    // shielded helion to proton mag. mom. ratio
    // Uncertainty: 8.9e-09
    fShieldedHelionToProtonMag_Mom_Ratio : LREAL := -0.7617665618;
    fShieldedHelionToProtonMag_Mom_Ratio_Uncertainty : LREAL := 8.9e-09;

    // shielded helion to shielded proton mag. mom. ratio
    // Uncertainty: 3.3e-09
    fShieldedHelionToShieldedProtonMag_Mom_Ratio : LREAL := -0.7617861313;
    fShieldedHelionToShieldedProtonMag_Mom_Ratio_Uncertainty : LREAL := 3.3e-09;

    // shielded proton gyromag. ratio (s^-1 T^-1)
    // Uncertainty: 2.9
    fShieldedProtonGyromag_Ratio_in_s_1_T_1 : LREAL := 267515315.1;
    fShieldedProtonGyromag_Ratio_in_s_1_T_1_Units : STRING := 's^-1 T^-1';
    fShieldedProtonGyromag_Ratio_in_s_1_T_1_Uncertainty : LREAL := 2.9;

    // shielded proton gyromag. ratio over 2 pi (MHz T^-1)
    // Uncertainty: 5.3e-07
    fShieldedProtonGyromag_RatioOver2Pi_in_MHz_T_1 : LREAL := 42.57638507;
    fShieldedProtonGyromag_RatioOver2Pi_in_MHz_T_1_Units : STRING := 'MHz T^-1';
    fShieldedProtonGyromag_RatioOver2Pi_in_MHz_T_1_Uncertainty : LREAL := 5.3e-07;

    // shielded proton mag. mom. (J T^-1)
    // Uncertainty: 1.5e-34
    fShieldedProtonMag_Mom_in_J_T_1 : LREAL := 1.41057056e-26;
    fShieldedProtonMag_Mom_in_J_T_1_Units : STRING := 'J T^-1';
    fShieldedProtonMag_Mom_in_J_T_1_Uncertainty : LREAL := 1.5e-34;

    // shielded proton mag. mom. to Bohr magneton ratio
    // Uncertainty: 1.7e-11
    fShieldedProtonMag_Mom_ToBohrMagnetonRatio : LREAL := 0.001520993128;
    fShieldedProtonMag_Mom_ToBohrMagnetonRatio_Uncertainty : LREAL := 1.7e-11;

    // shielded proton mag. mom. to nuclear magneton ratio
    // Uncertainty: 3e-08
    fShieldedProtonMag_Mom_ToNuclearMagnetonRatio : LREAL := 2.792775599;
    fShieldedProtonMag_Mom_ToNuclearMagnetonRatio_Uncertainty : LREAL := 3e-08;

    // speed of light in vacuum (m s^-1)
    fSpeedOfLightInVacuum_in_m_s_1 : LREAL := 299792458.0;
    fSpeedOfLightInVacuum_in_m_s_1_Units : STRING := 'm s^-1';

    // standard acceleration of gravity (m s^-2)
    fStandardAccelerationOfGravity_in_m_s_2 : LREAL := 9.80665;
    fStandardAccelerationOfGravity_in_m_s_2_Units : STRING := 'm s^-2';

    // standard atmosphere (Pa)
    fStandardAtmosphere_in_Pa : LREAL := 101325.0;
    fStandardAtmosphere_in_Pa_Units : STRING := 'Pa';

    // Stefan-Boltzmann constant (W m^-2 K^-4)
    fStefan_BoltzmannConstant_in_W_m_2_K_4 : LREAL := 5.670374419e-08;
    fStefan_BoltzmannConstant_in_W_m_2_K_4_Units : STRING := 'W m^-2 K^-4';

    // tau Compton wavelength (m)
    // Uncertainty: 4.7e-20
    fTauComptonWavelength_in_m : LREAL := 6.97771e-16;
    fTauComptonWavelength_in_m_Units : STRING := 'm';
    fTauComptonWavelength_in_m_Uncertainty : LREAL := 4.7e-20;

    // tau Compton wavelength over 2 pi (m)
    // Uncertainty: 1e-20
    fTauComptonWavelengthOver2Pi_in_m : LREAL := 1.11056e-16;
    fTauComptonWavelengthOver2Pi_in_m_Units : STRING := 'm';
    fTauComptonWavelengthOver2Pi_in_m_Uncertainty : LREAL := 1e-20;

    // tau-electron mass ratio
    // Uncertainty: 0.23
    fTauElectronMassRatio : LREAL := 3477.23;
    fTauElectronMassRatio_Uncertainty : LREAL := 0.23;

    // tau mass (kg)
    // Uncertainty: 2.1e-31
    fTauMass_in_kg : LREAL := 3.16754e-27;
    fTauMass_in_kg_Units : STRING := 'kg';
    fTauMass_in_kg_Uncertainty : LREAL := 2.1e-31;

    // tau mass energy equivalent (J)
    // Uncertainty: 1.9e-14
    fTauMassEnergyEquivalent_in_J : LREAL := 2.84684e-10;
    fTauMassEnergyEquivalent_in_J_Units : STRING := 'J';
    fTauMassEnergyEquivalent_in_J_Uncertainty : LREAL := 1.9e-14;

    // tau mass energy equivalent in MeV (MeV)
    // Uncertainty: 0.16
    fTauMassEnergyEquivalentInMeV_in_MeV : LREAL := 1776.82;
    fTauMassEnergyEquivalentInMeV_in_MeV_Units : STRING := 'MeV';
    fTauMassEnergyEquivalentInMeV_in_MeV_Uncertainty : LREAL := 0.16;

    // tau mass in u (u)
    // Uncertainty: 0.00013
    fTauMassInU_in_u : LREAL := 1.90754;
    fTauMassInU_in_u_Units : STRING := 'u';
    fTauMassInU_in_u_Uncertainty : LREAL := 0.00013;

    // tau molar mass (kg mol^-1)
    // Uncertainty: 1.3e-07
    fTauMolarMass_in_kg_mol_1 : LREAL := 0.00190754;
    fTauMolarMass_in_kg_mol_1_Units : STRING := 'kg mol^-1';
    fTauMolarMass_in_kg_mol_1_Uncertainty : LREAL := 1.3e-07;

    // tau-muon mass ratio
    // Uncertainty: 0.0011
    fTauMuonMassRatio : LREAL := 16.817;
    fTauMuonMassRatio_Uncertainty : LREAL := 0.0011;

    // tau-neutron mass ratio
    // Uncertainty: 0.00013
    fTauNeutronMassRatio : LREAL := 1.89115;
    fTauNeutronMassRatio_Uncertainty : LREAL := 0.00013;

    // tau-proton mass ratio
    // Uncertainty: 0.00013
    fTauProtonMassRatio : LREAL := 1.89376;
    fTauProtonMassRatio_Uncertainty : LREAL := 0.00013;

    // Thomson cross section (m^2)
    // Uncertainty: 6e-38
    fThomsonCrossSection_in_m_2 : LREAL := 6.6524587321e-29;
    fThomsonCrossSection_in_m_2_Units : STRING := 'm^2';
    fThomsonCrossSection_in_m_2_Uncertainty : LREAL := 6e-38;

    // triton-electron mag. mom. ratio
    // Uncertainty: 2.1e-11
    fTritonElectronMag_Mom_Ratio : LREAL := -0.001620514423;
    fTritonElectronMag_Mom_Ratio_Uncertainty : LREAL := 2.1e-11;

    // triton-electron mass ratio
    // Uncertainty: 2.7e-07
    fTritonElectronMassRatio : LREAL := 5496.92153573;
    fTritonElectronMassRatio_Uncertainty : LREAL := 2.7e-07;

    // triton g factor
    // Uncertainty: 1.2e-08
    fTritonGFactor : LREAL := 5.957924931;
    fTritonGFactor_Uncertainty : LREAL := 1.2e-08;

    // triton mag. mom. (J T^-1)
    // Uncertainty: 3e-35
    fTritonMag_Mom_in_J_T_1 : LREAL := 1.5046095202e-26;
    fTritonMag_Mom_in_J_T_1_Units : STRING := 'J T^-1';
    fTritonMag_Mom_in_J_T_1_Uncertainty : LREAL := 3e-35;

    // triton mag. mom. to Bohr magneton ratio
    // Uncertainty: 3.2e-12
    fTritonMag_Mom_ToBohrMagnetonRatio : LREAL := 0.0016223936651;
    fTritonMag_Mom_ToBohrMagnetonRatio_Uncertainty : LREAL := 3.2e-12;

    // triton mag. mom. to nuclear magneton ratio
    // Uncertainty: 5.9e-09
    fTritonMag_Mom_ToNuclearMagnetonRatio : LREAL := 2.9789624656;
    fTritonMag_Mom_ToNuclearMagnetonRatio_Uncertainty : LREAL := 5.9e-09;

    // triton mass (kg)
    // Uncertainty: 1.5e-36
    fTritonMass_in_kg : LREAL := 5.0073567446e-27;
    fTritonMass_in_kg_Units : STRING := 'kg';
    fTritonMass_in_kg_Uncertainty : LREAL := 1.5e-36;

    // triton mass energy equivalent (J)
    // Uncertainty: 1.4e-19
    fTritonMassEnergyEquivalent_in_J : LREAL := 4.500387806e-10;
    fTritonMassEnergyEquivalent_in_J_Units : STRING := 'J';
    fTritonMassEnergyEquivalent_in_J_Uncertainty : LREAL := 1.4e-19;

    // triton mass energy equivalent in MeV (MeV)
    // Uncertainty: 8.5e-07
    fTritonMassEnergyEquivalentInMeV_in_MeV : LREAL := 2808.92113298;
    fTritonMassEnergyEquivalentInMeV_in_MeV_Units : STRING := 'MeV';
    fTritonMassEnergyEquivalentInMeV_in_MeV_Uncertainty : LREAL := 8.5e-07;

    // triton mass in u (u)
    // Uncertainty: 1.2e-10
    fTritonMassInU_in_u : LREAL := 3.01550071621;
    fTritonMassInU_in_u_Units : STRING := 'u';
    fTritonMassInU_in_u_Uncertainty : LREAL := 1.2e-10;

    // triton molar mass (kg mol^-1)
    // Uncertainty: 9.2e-13
    fTritonMolarMass_in_kg_mol_1 : LREAL := 0.00301550071517;
    fTritonMolarMass_in_kg_mol_1_Units : STRING := 'kg mol^-1';
    fTritonMolarMass_in_kg_mol_1_Uncertainty : LREAL := 9.2e-13;

    // triton-neutron mag. mom. ratio
    // Uncertainty: 3.7e-07
    fTritonNeutronMag_Mom_Ratio : LREAL := -1.55718553;
    fTritonNeutronMag_Mom_Ratio_Uncertainty : LREAL := 3.7e-07;

    // triton-proton mag. mom. ratio
    // Uncertainty: 1e-08
    fTritonProtonMag_Mom_Ratio : LREAL := 1.066639908;
    fTritonProtonMag_Mom_Ratio_Uncertainty : LREAL := 1e-08;

    // triton-proton mass ratio
    // Uncertainty: 1.5e-10
    fTritonProtonMassRatio : LREAL := 2.99371703414;
    fTritonProtonMassRatio_Uncertainty : LREAL := 1.5e-10;

    // unified atomic mass unit (kg)
    // Uncertainty: 5e-37
    fUnifiedAtomicMassUnit_in_kg : LREAL := 1.6605390666e-27;
    fUnifiedAtomicMassUnit_in_kg_Units : STRING := 'kg';
    fUnifiedAtomicMassUnit_in_kg_Uncertainty : LREAL := 5e-37;

    // von Klitzing constant (ohm)
    fVonKlitzingConstant_in_ohm : LREAL := 25812.80745;
    fVonKlitzingConstant_in_ohm_Units : STRING := 'ohm';

    // weak mixing angle
    // Uncertainty: 0.0003
    fWeakMixingAngle : LREAL := 0.2229;
    fWeakMixingAngle_Uncertainty : LREAL := 0.0003;

    // Wien frequency displacement law constant (Hz K^-1)
    fWienFrequencyDisplacementLawConstant_in_Hz_K_1 : LREAL := 58789257570.0;
    fWienFrequencyDisplacementLawConstant_in_Hz_K_1_Units : STRING := 'Hz K^-1';

    // Wien wavelength displacement law constant (m K)
    fWienWavelengthDisplacementLawConstant_in_m_K : LREAL := 0.002897771955;
    fWienWavelengthDisplacementLawConstant_in_m_K_Units : STRING := 'm K';

    // atomic unit of mom.um (kg m s^-1)
    // Uncertainty: 2.4e-32
    fAtomicUnitOfMom_um_in_kg_m_s_1 : LREAL := 1.992851882e-24;
    fAtomicUnitOfMom_um_in_kg_m_s_1_Units : STRING := 'kg m s^-1';
    fAtomicUnitOfMom_um_in_kg_m_s_1_Uncertainty : LREAL := 2.4e-32;

    // electron-helion mass ratio
    // Uncertainty: 7.9e-15
    fElectronHelionMassRatio : LREAL := 0.0001819543074573;
    fElectronHelionMassRatio_Uncertainty : LREAL := 7.9e-15;

    // electron-triton mass ratio
    // Uncertainty: 9e-15
    fElectronTritonMassRatio : LREAL := 0.0001819200062251;
    fElectronTritonMassRatio_Uncertainty : LREAL := 9e-15;

    // helion g factor
    // Uncertainty: 5e-08
    fHelionGFactor : LREAL := -4.255250615;
    fHelionGFactor_Uncertainty : LREAL := 5e-08;

    // helion mag. mom. (J T^-1)
    // Uncertainty: 1.3e-34
    fHelionMag_Mom_in_J_T_1 : LREAL := -1.074617532e-26;
    fHelionMag_Mom_in_J_T_1_Units : STRING := 'J T^-1';
    fHelionMag_Mom_in_J_T_1_Uncertainty : LREAL := 1.3e-34;

    // helion mag. mom. to Bohr magneton ratio
    // Uncertainty: 1.4e-11
    fHelionMag_Mom_ToBohrMagnetonRatio : LREAL := -0.001158740958;
    fHelionMag_Mom_ToBohrMagnetonRatio_Uncertainty : LREAL := 1.4e-11;

    // helion mag. mom. to nuclear magneton ratio
    // Uncertainty: 2.5e-08
    fHelionMag_Mom_ToNuclearMagnetonRatio : LREAL := -2.127625307;
    fHelionMag_Mom_ToNuclearMagnetonRatio_Uncertainty : LREAL := 2.5e-08;

    // Loschmidt constant (273.15 K, 100 kPa) (m^-3)
    fLoschmidtConstant_273_15K_100KPa_in_m_3 : LREAL := 2.651645804e+25;
    fLoschmidtConstant_273_15K_100KPa_in_m_3_Units : STRING := 'm^-3';

    // natural unit of mom.um (kg m s^-1)
    // Uncertainty: 3.4e-30
    fNaturalUnitOfMom_um_in_kg_m_s_1 : LREAL := 2.730924488e-22;
    fNaturalUnitOfMom_um_in_kg_m_s_1_Units : STRING := 'kg m s^-1';
    fNaturalUnitOfMom_um_in_kg_m_s_1_Uncertainty : LREAL := 3.4e-30;

    // natural unit of mom.um in MeV/c (MeV/c)
    // Uncertainty: 3.1e-09
    fNaturalUnitOfMom_umInMeV_c_in_MeV_c : LREAL := 0.5109989461;
    fNaturalUnitOfMom_umInMeV_c_in_MeV_c_Units : STRING := 'MeV/c';
    fNaturalUnitOfMom_umInMeV_c_in_MeV_c_Uncertainty : LREAL := 3.1e-09;

    // neutron-proton mass difference (kg)
    // Uncertainty: 8.2e-37
    fNeutronProtonMassDifference_in_kg : LREAL := 2.30557435e-30;
    fNeutronProtonMassDifference_in_kg_Units : STRING := 'kg';
    fNeutronProtonMassDifference_in_kg_Uncertainty : LREAL := 8.2e-37;

    // neutron-proton mass difference energy equivalent (J)
    // Uncertainty: 7.4e-20
    fNeutronProtonMassDifferenceEnergyEquivalent_in_J : LREAL := 2.07214689e-13;
    fNeutronProtonMassDifferenceEnergyEquivalent_in_J_Units : STRING := 'J';
    fNeutronProtonMassDifferenceEnergyEquivalent_in_J_Uncertainty : LREAL := 7.4e-20;

    // neutron-proton mass difference energy equivalent in MeV (MeV)
    // Uncertainty: 4.6e-07
    fNeutronProtonMassDifferenceEnergyEquivalentInMeV_in_MeV : LREAL := 1.29333236;
    fNeutronProtonMassDifferenceEnergyEquivalentInMeV_in_MeV_Units : STRING := 'MeV';
    fNeutronProtonMassDifferenceEnergyEquivalentInMeV_in_MeV_Uncertainty : LREAL := 4.6e-07;

    // neutron-proton mass difference in u (u)
    // Uncertainty: 4.9e-10
    fNeutronProtonMassDifferenceInU_in_u : LREAL := 0.00138844933;
    fNeutronProtonMassDifferenceInU_in_u_Units : STRING := 'u';
    fNeutronProtonMassDifferenceInU_in_u_Uncertainty : LREAL := 4.9e-10;

    // standard-state pressure (Pa)
    fStandardStatePressure_in_Pa : LREAL := 100000.0;
    fStandardStatePressure_in_Pa_Units : STRING := 'Pa';

    // alpha particle relative atomic mass
    // Uncertainty: 6.3e-11
    fAlphaParticleRelativeAtomicMass : LREAL := 4.001506179127;
    fAlphaParticleRelativeAtomicMass_Uncertainty : LREAL := 6.3e-11;

    // Bohr magneton in inverse meter per tesla (m^-1 T^-1)
    // Uncertainty: 1.4e-08
    fBohrMagnetonInInverseMeterPerTesla_in_m_1_T_1 : LREAL := 46.686447783;
    fBohrMagnetonInInverseMeterPerTesla_in_m_1_T_1_Units : STRING := 'm^-1 T^-1';
    fBohrMagnetonInInverseMeterPerTesla_in_m_1_T_1_Uncertainty : LREAL := 1.4e-08;

    // Boltzmann constant in inverse meter per kelvin (m^-1 K^-1)
    fBoltzmannConstantInInverseMeterPerKelvin_in_m_1_K_1 : LREAL := 69.50348004;
    fBoltzmannConstantInInverseMeterPerKelvin_in_m_1_K_1_Units : STRING := 'm^-1 K^-1';

    // conventional value of ampere-90 (A)
    fConventionalValueOfAmpere_90_in_A : LREAL := 1.00000008887;
    fConventionalValueOfAmpere_90_in_A_Units : STRING := 'A';

    // conventional value of coulomb-90 (C)
    fConventionalValueOfCoulomb_90_in_C : LREAL := 1.00000008887;
    fConventionalValueOfCoulomb_90_in_C_Units : STRING := 'C';

    // conventional value of farad-90 (F)
    fConventionalValueOfFarad_90_in_F : LREAL := 0.9999999822;
    fConventionalValueOfFarad_90_in_F_Units : STRING := 'F';

    // conventional value of henry-90 (H)
    fConventionalValueOfHenry_90_in_H : LREAL := 1.00000001779;
    fConventionalValueOfHenry_90_in_H_Units : STRING := 'H';

    // conventional value of ohm-90 (ohm)
    fConventionalValueOfOhm_90_in_ohm : LREAL := 1.00000001779;
    fConventionalValueOfOhm_90_in_ohm_Units : STRING := 'ohm';

    // conventional value of volt-90 (V)
    fConventionalValueOfVolt_90_in_V : LREAL := 1.00000010666;
    fConventionalValueOfVolt_90_in_V_Units : STRING := 'V';

    // conventional value of watt-90 (W)
    fConventionalValueOfWatt_90_in_W : LREAL := 1.00000019553;
    fConventionalValueOfWatt_90_in_W_Units : STRING := 'W';

    // deuteron relative atomic mass
    // Uncertainty: 4e-11
    fDeuteronRelativeAtomicMass : LREAL := 2.013553212745;
    fDeuteronRelativeAtomicMass_Uncertainty : LREAL := 4e-11;

    // electron gyromag. ratio in MHz/T (MHz T^-1)
    // Uncertainty: 8.5e-06
    fElectronGyromag_RatioInMHz_T_in_MHz_T_1 : LREAL := 28024.9514242;
    fElectronGyromag_RatioInMHz_T_in_MHz_T_1_Units : STRING := 'MHz T^-1';
    fElectronGyromag_RatioInMHz_T_in_MHz_T_1_Uncertainty : LREAL := 8.5e-06;

    // electron relative atomic mass
    // Uncertainty: 1.6e-14
    fElectronRelativeAtomicMass : LREAL := 0.000548579909065;
    fElectronRelativeAtomicMass_Uncertainty : LREAL := 1.6e-14;

    // elementary charge over h-bar (A J^-1)
    fElementaryChargeOverH_bar_in_A_J_1 : LREAL := 1519267447000000.0;
    fElementaryChargeOverH_bar_in_A_J_1_Units : STRING := 'A J^-1';

    // helion relative atomic mass
    // Uncertainty: 9.7e-11
    fHelionRelativeAtomicMass : LREAL := 3.014932247175;
    fHelionRelativeAtomicMass_Uncertainty : LREAL := 9.7e-11;

    // helion shielding shift
    // Uncertainty: 1e-10
    fHelionShieldingShift : LREAL := 5.996743e-05;
    fHelionShieldingShift_Uncertainty : LREAL := 1e-10;

    // hyperfine transition frequency of Cs-133 (Hz)
    fHyperfineTransitionFrequencyOfCs_133_in_Hz : LREAL := 9192631770.0;
    fHyperfineTransitionFrequencyOfCs_133_in_Hz_Units : STRING := 'Hz';

    // lattice spacing of ideal Si (220) (m)
    // Uncertainty: 3.2e-18
    fLatticeSpacingOfIdealSi_220_in_m : LREAL := 1.920155716e-10;
    fLatticeSpacingOfIdealSi_220_in_m_Units : STRING := 'm';
    fLatticeSpacingOfIdealSi_220_in_m_Uncertainty : LREAL := 3.2e-18;

    // luminous efficacy (lm W^-1)
    fLuminousEfficacy_in_lm_W_1 : LREAL := 683.0;
    fLuminousEfficacy_in_lm_W_1_Units : STRING := 'lm W^-1';

    // neutron gyromag. ratio in MHz/T (MHz T^-1)
    // Uncertainty: 6.9e-06
    fNeutronGyromag_RatioInMHz_T_in_MHz_T_1 : LREAL := 29.1646931;
    fNeutronGyromag_RatioInMHz_T_in_MHz_T_1_Units : STRING := 'MHz T^-1';
    fNeutronGyromag_RatioInMHz_T_in_MHz_T_1_Uncertainty : LREAL := 6.9e-06;

    // neutron relative atomic mass
    // Uncertainty: 4.9e-10
    fNeutronRelativeAtomicMass : LREAL := 1.00866491595;
    fNeutronRelativeAtomicMass_Uncertainty : LREAL := 4.9e-10;

    // nuclear magneton in inverse meter per tesla (m^-1 T^-1)
    // Uncertainty: 7.8e-12
    fNuclearMagnetonInInverseMeterPerTesla_in_m_1_T_1 : LREAL := 0.0254262341353;
    fNuclearMagnetonInInverseMeterPerTesla_in_m_1_T_1_Units : STRING := 'm^-1 T^-1';
    fNuclearMagnetonInInverseMeterPerTesla_in_m_1_T_1_Uncertainty : LREAL := 7.8e-12;

    // Planck constant in eV/Hz (eV Hz^-1)
    fPlanckConstantInEV_Hz_in_eV_Hz_1 : LREAL := 4.135667696e-15;
    fPlanckConstantInEV_Hz_in_eV_Hz_1_Units : STRING := 'eV Hz^-1';

    // proton gyromag. ratio in MHz/T (MHz T^-1)
    // Uncertainty: 1.8e-08
    fProtonGyromag_RatioInMHz_T_in_MHz_T_1 : LREAL := 42.577478518;
    fProtonGyromag_RatioInMHz_T_in_MHz_T_1_Units : STRING := 'MHz T^-1';
    fProtonGyromag_RatioInMHz_T_in_MHz_T_1_Uncertainty : LREAL := 1.8e-08;

    // proton relative atomic mass
    // Uncertainty: 5.3e-11
    fProtonRelativeAtomicMass : LREAL := 1.007276466621;
    fProtonRelativeAtomicMass_Uncertainty : LREAL := 5.3e-11;

    // reduced Compton wavelength (m)
    // Uncertainty: 1.2e-22
    fReducedComptonWavelength_in_m : LREAL := 3.8615926796e-13;
    fReducedComptonWavelength_in_m_Units : STRING := 'm';
    fReducedComptonWavelength_in_m_Uncertainty : LREAL := 1.2e-22;

    // reduced muon Compton wavelength (m)
    // Uncertainty: 4.2e-23
    fReducedMuonComptonWavelength_in_m : LREAL := 1.867594306e-15;
    fReducedMuonComptonWavelength_in_m_Units : STRING := 'm';
    fReducedMuonComptonWavelength_in_m_Uncertainty : LREAL := 4.2e-23;

    // reduced neutron Compton wavelength (m)
    // Uncertainty: 1.2e-25
    fReducedNeutronComptonWavelength_in_m : LREAL := 2.1001941552e-16;
    fReducedNeutronComptonWavelength_in_m_Units : STRING := 'm';
    fReducedNeutronComptonWavelength_in_m_Uncertainty : LREAL := 1.2e-25;

    // reduced Planck constant (J s)
    fReducedPlanckConstant_in_J_s : LREAL := 1.054571817e-34;
    fReducedPlanckConstant_in_J_s_Units : STRING := 'J s';

    // reduced Planck constant in eV s (eV s)
    fReducedPlanckConstantInEVS_in_eV_s : LREAL := 6.582119569e-16;
    fReducedPlanckConstantInEVS_in_eV_s_Units : STRING := 'eV s';

    // reduced Planck constant times c in MeV fm (MeV fm)
    fReducedPlanckConstantTimesCInMeVFm_in_MeV_fm : LREAL := 197.3269804;
    fReducedPlanckConstantTimesCInMeVFm_in_MeV_fm_Units : STRING := 'MeV fm';

    // reduced proton Compton wavelength (m)
    // Uncertainty: 6.4e-26
    fReducedProtonComptonWavelength_in_m : LREAL := 2.10308910336e-16;
    fReducedProtonComptonWavelength_in_m_Units : STRING := 'm';
    fReducedProtonComptonWavelength_in_m_Uncertainty : LREAL := 6.4e-26;

    // reduced tau Compton wavelength (m)
    // Uncertainty: 7.5e-21
    fReducedTauComptonWavelength_in_m : LREAL := 1.110538e-16;
    fReducedTauComptonWavelength_in_m_Units : STRING := 'm';
    fReducedTauComptonWavelength_in_m_Uncertainty : LREAL := 7.5e-21;

    // shielded helion gyromag. ratio in MHz/T (MHz T^-1)
    // Uncertainty: 3.8e-07
    fShieldedHelionGyromag_RatioInMHz_T_in_MHz_T_1 : LREAL := 32.43409942;
    fShieldedHelionGyromag_RatioInMHz_T_in_MHz_T_1_Units : STRING := 'MHz T^-1';
    fShieldedHelionGyromag_RatioInMHz_T_in_MHz_T_1_Uncertainty : LREAL := 3.8e-07;

    // shielded proton gyromag. ratio in MHz/T (MHz T^-1)
    // Uncertainty: 4.6e-07
    fShieldedProtonGyromag_RatioInMHz_T_in_MHz_T_1 : LREAL := 42.57638474;
    fShieldedProtonGyromag_RatioInMHz_T_in_MHz_T_1_Units : STRING := 'MHz T^-1';
    fShieldedProtonGyromag_RatioInMHz_T_in_MHz_T_1_Uncertainty : LREAL := 4.6e-07;

    // shielding difference of d and p in HD
    // Uncertainty: 2e-11
    fShieldingDifferenceOfDAndPInHD : LREAL := 2.02e-08;
    fShieldingDifferenceOfDAndPInHD_Uncertainty : LREAL := 2e-11;

    // shielding difference of t and p in HT
    // Uncertainty: 2e-11
    fShieldingDifferenceOfTAndPInHT : LREAL := 2.414e-08;
    fShieldingDifferenceOfTAndPInHT_Uncertainty : LREAL := 2e-11;

    // tau energy equivalent (MeV)
    // Uncertainty: 0.12
    fTauEnergyEquivalent_in_MeV : LREAL := 1776.86;
    fTauEnergyEquivalent_in_MeV_Units : STRING := 'MeV';
    fTauEnergyEquivalent_in_MeV_Uncertainty : LREAL := 0.12;

    // triton relative atomic mass
    // Uncertainty: 1.2e-10
    fTritonRelativeAtomicMass : LREAL := 3.01550071621;
    fTritonRelativeAtomicMass_Uncertainty : LREAL := 1.2e-10;

    // triton to proton mag. mom. ratio
    // Uncertainty: 2.1e-09
    fTritonToProtonMag_Mom_Ratio : LREAL := 1.0666399191;
    fTritonToProtonMag_Mom_Ratio_Uncertainty : LREAL := 2.1e-09;

    // vacuum electric permittivity (F m^-1)
    // Uncertainty: 1.3e-21
    fVacuumElectricPermittivity_in_F_m_1 : LREAL := 8.8541878128e-12;
    fVacuumElectricPermittivity_in_F_m_1_Units : STRING := 'F m^-1';
    fVacuumElectricPermittivity_in_F_m_1_Uncertainty : LREAL := 1.3e-21;

    // vacuum mag. permeability (N A^-2)
    // Uncertainty: 1.9e-16
    fVacuumMag_Permeability_in_N_A_2 : LREAL := 1.25663706212e-06;
    fVacuumMag_Permeability_in_N_A_2_Units : STRING := 'N A^-2';
    fVacuumMag_Permeability_in_N_A_2_Uncertainty : LREAL := 1.9e-16;

    // W to Z mass ratio
    // Uncertainty: 0.00017
    fWToZMassRatio : LREAL := 0.88153;
    fWToZMassRatio_Uncertainty : LREAL := 0.00017;

END_VAR

// ---- GVLs/GVL_Physics.TcGVL
{attribute 'qualified_only'}
VAR_GLOBAL
    fbScatteringFactors : FB_ScatteringFactorLUT;
END_VAR
VAR_GLOBAL CONSTANT
    nMaxNumLensesInSet : INT := 10;
END_VAR

// ---- ITFs/I_ScatteringFactorLookup.TcIO
INTERFACE I_ScatteringFactorLookup


METHOD GetScatteringFactor
VAR_INPUT
    sMaterialName : T_MaxString; (* Chemical formula for the material as a string. *)
    fPhotonEnergy_eV : LREAL; (* Photon energy in eV. *)
END_VAR
VAR_OUTPUT
    f1 : LREAL;
    f2 : LREAL;
    bError : BOOL;
    sErrorMsg : T_MaxString;
END_VAR
END_METHOD

PROPERTY MaximumValidLookupPhotonEnergy_eV : LREAL
GET
END_GET
END_PROPERTY

PROPERTY MinimumValidLookupPhotonEnergy_eV : LREAL
GET
END_GET
END_PROPERTY

END_INTERFACE

// ---- POUs/RunTests.TcPOU

PROGRAM RunTests
VAR
    fbAtomicMassLookup_Test : FB_AtomicMassLookup_Test;
    fbAtomicNumberLookup_Test : FB_AtomicNumberLookup_Test;
    fbCalculateMassAttenuationCoefficient_Test : FB_CalculateXrayAbsorptionConstant_Test;
    fbCalculateThicknessFromTransmission_Test : FB_CalculateThicknessFromTransmission_Test;
    fbMaterialDensityLookup_Test : FB_MaterialDensityLookup_Test;
    fbScatteringFactorLookupCXRO_Test : FB_ScatteringFactorLookupCXRO_Test;
    fbScatteringFactorLUT_Test : FB_ScatteringFactorLUT_Test;
    fbTestTransmission : FB_TestTransmission;
    fbTestElementDensity : FB_TestElementDensity;
    fbAtomicNumber_Test : FB_AtomicNumber_Test;

    (* Smoke test - just instantiate *)
    fbPhysicalConstants : FB_PhysicalConstants;
    fbAtomicMass : FB_AtomicMass;

END_VAR


TcUnit.RUN();

fbPhysicalConstants();
fbAtomicMass();

END_PROGRAM

// ---- Tests/FB_AtomicMassLookup_Test.TcPOU

FUNCTION_BLOCK FB_AtomicMassLookup_Test EXTENDS TcUnit.FB_TestSuite
VAR
END_VAR


GivenElementExpectCorrectAtomicMass();


METHOD PRIVATE GivenElementExpectCorrectAtomicMass
VAR
    fResult : LREAL;
END_VAR

TEST('GivenElementExpectCorrectAtomicMass');

fResult := F_AtomicMassLookup(
    sMaterialName := 'C'
);

AssertEquals_LREAL(
    Expected := 12.0107,
    Actual := fResult,
    Delta := 1e-9,
    Message := 'Incorrect result.'
);

fResult := F_AtomicMassLookup(
    sMaterialName := 'Co'
);

AssertEquals_LREAL(
    Expected := 58.9332,
    Actual := fResult,
    Delta := 1e-9,
    Message := 'Incorrect result.'
);

fResult := F_AtomicMassLookup(
    sMaterialName := 'Cd'
);

AssertEquals_LREAL(
    Expected := 112.411,
    Actual := fResult,
    Delta := 1e-9,
    Message := 'Incorrect result.'
);

TEST_FINISHED();
END_METHOD

END_FUNCTION_BLOCK

// ---- POUs/F_AtomicMassLookup.TcPOU

FUNCTION F_AtomicMassLookup : LREAL
VAR_INPUT
    sMaterialName : T_MaxString;
END_VAR
VAR
    fbAtomicMass : FB_AtomicMass;
END_VAR


fbAtomicMass(
    sName := sMaterialName
);

IF fbAtomicMass.bFound THEN
    F_AtomicMassLookup := fbAtomicMass.fValue;
ELSE
    F_AtomicMassLookup := -1.0;
END_IF

END_FUNCTION

// ---- POUs/FB_AtomicMass.TcPOU

(* WARNING: This file is auto-generated. Do not modify it.*)
FUNCTION_BLOCK FB_AtomicMass

VAR_INPUT
    sName : STRING;
END_VAR

VAR_OUTPUT
    bFound : BOOL;
    fValue : LREAL;
    fUncertainty : LREAL;
    sDescription : STRING;
    sUnits : STRING;
    sCaveat : STRING;
END_VAR


(* WARNING: This file is auto-generated. Do not modify it.*)
IF sName = 'n' THEN
    fValue := 1.00866491597;
    fUncertainty := 0;
    sDescription := 'Atomic mass of n (neutron)';
    sUnits := 'None';
    sCaveat := 'None';
    bFound := TRUE;
ELSIF sName = 'H' THEN
    fValue := 1.00794;
    fUncertainty := 0;
    sDescription := 'Atomic mass of H (hydrogen)';
    sUnits := 'None';
    sCaveat := 'None';
    bFound := TRUE;
ELSIF sName = 'He' THEN
    fValue := 4.002602;
    fUncertainty := 0;
    sDescription := 'Atomic mass of He (helium)';
    sUnits := 'None';
    sCaveat := 'None';
    bFound := TRUE;
ELSIF sName = 'Li' THEN
    fValue := 6.941;
    fUncertainty := 0;
    sDescription := 'Atomic mass of Li (lithium)';
    sUnits := 'None';
    sCaveat := 'None';
    bFound := TRUE;
ELSIF sName = 'Be' THEN
    fValue := 9.012182;
    fUncertainty := 0;
    sDescription := 'Atomic mass of Be (beryllium)';
    sUnits := 'None';
    sCaveat := 'None';
    bFound := TRUE;
ELSIF sName = 'B' THEN
    fValue := 10.811;
    fUncertainty := 0;
    sDescription := 'Atomic mass of B (boron)';
    sUnits := 'None';
    sCaveat := 'None';
    bFound := TRUE;
ELSIF sName = 'C' OR sName = 'C (Diamond)' THEN
    fValue := 12.0107;
    fUncertainty := 0;
    sDescription := 'Atomic mass of C (carbon)';
    sUnits := 'None';
    sCaveat := 'None';
    bFound := TRUE;
ELSIF sName = 'N' THEN
    fValue := 14.0067;
    fUncertainty := 0;
    sDescription := 'Atomic mass of N (nitrogen)';
    sUnits := 'None';
    sCaveat := 'None';
    bFound := TRUE;
ELSIF sName = 'O' THEN
    fValue := 15.9994;
    fUncertainty := 0;
    sDescription := 'Atomic mass of O (oxygen)';
    sUnits := 'None';
    sCaveat := 'None';
    bFound := TRUE;
ELSIF sName = 'F' THEN
    fValue := 18.9984032;
    fUncertainty := 0;
    sDescription := 'Atomic mass of F (fluorine)';
    sUnits := 'None';
    sCaveat := 'None';
    bFound := TRUE;
ELSIF sName = 'Ne' THEN
    fValue := 20.1797;
    fUncertainty := 0;
    sDescription := 'Atomic mass of Ne (neon)';
    sUnits := 'None';
    sCaveat := 'None';
    bFound := TRUE;
ELSIF sName = 'Na' THEN
    fValue := 22.98977;
    fUncertainty := 0;
    sDescription := 'Atomic mass of Na (sodium)';
    sUnits := 'None';
    sCaveat := 'None';
    bFound := TRUE;
ELSIF sName = 'Mg' THEN
    fValue := 24.305;
    fUncertainty := 0;
    sDescription := 'Atomic mass of Mg (magnesium)';
    sUnits := 'None';
    sCaveat := 'None';
    bFound := TRUE;
ELSIF sName = 'Al' THEN
    fValue := 26.981538;
    fUncertainty := 0;
    sDescription := 'Atomic mass of Al (aluminum)';
    sUnits := 'None';
    sCaveat := 'None';
    bFound := TRUE;
ELSIF sName = 'Si' THEN
    fValue := 28.0855;
    fUncertainty := 0;
    sDescription := 'Atomic mass of Si (silicon)';
    sUnits := 'None';
    sCaveat := 'None';
    bFound := TRUE;
ELSIF sName = 'P' THEN
    fValue := 30.973761;
    fUncertainty := 0;
    sDescription := 'Atomic mass of P (phosphorus)';
    sUnits := 'None';
    sCaveat := 'None';
    bFound := TRUE;
ELSIF sName = 'S' THEN
    fValue := 32.065;
    fUncertainty := 0;
    sDescription := 'Atomic mass of S (sulfur)';
    sUnits := 'None';
    sCaveat := 'None';
    bFound := TRUE;
ELSIF sName = 'Cl' THEN
    fValue := 35.453;
    fUncertainty := 0;
    sDescription := 'Atomic mass of Cl (chlorine)';
    sUnits := 'None';
    sCaveat := 'None';
    bFound := TRUE;
ELSIF sName = 'Ar' THEN
    fValue := 39.948;
    fUncertainty := 0;
    sDescription := 'Atomic mass of Ar (argon)';
    sUnits := 'None';
    sCaveat := 'None';
    bFound := TRUE;
ELSIF sName = 'K' THEN
    fValue := 39.0983;
    fUncertainty := 0;
    sDescription := 'Atomic mass of K (potassium)';
    sUnits := 'None';
    sCaveat := 'None';
    bFound := TRUE;
ELSIF sName = 'Ca' THEN
    fValue := 40.078;
    fUncertainty := 0;
    sDescription := 'Atomic mass of Ca (calcium)';
    sUnits := 'None';
    sCaveat := 'None';
    bFound := TRUE;
ELSIF sName = 'Sc' THEN
    fValue := 44.95591;
    fUncertainty := 0;
    sDescription := 'Atomic mass of Sc (scandium)';
    sUnits := 'None';
    sCaveat := 'None';
    bFound := TRUE;
ELSIF sName = 'Ti' THEN
    fValue := 47.867;
    fUncertainty := 0;
    sDescription := 'Atomic mass of Ti (titanium)';
    sUnits := 'None';
    sCaveat := 'None';
    bFound := TRUE;
ELSIF sName = 'V' THEN
    fValue := 50.9415;
    fUncertainty := 0;
    sDescription := 'Atomic mass of V (vanadium)';
    sUnits := 'None';
    sCaveat := 'None';
    bFound := TRUE;
ELSIF sName = 'Cr' THEN
    fValue := 51.9961;
    fUncertainty := 0;
    sDescription := 'Atomic mass of Cr (chromium)';
    sUnits := 'None';
    sCaveat := 'None';
    bFound := TRUE;
ELSIF sName = 'Mn' THEN
    fValue := 54.938049;
    fUncertainty := 0;
    sDescription := 'Atomic mass of Mn (manganese)';
    sUnits := 'None';
    sCaveat := 'None';
    bFound := TRUE;
ELSIF sName = 'Fe' THEN
    fValue := 55.845;
    fUncertainty := 0;
    sDescription := 'Atomic mass of Fe (iron)';
    sUnits := 'None';
    sCaveat := 'None';
    bFound := TRUE;
ELSIF sName = 'Co' THEN
    fValue := 58.9332;
    fUncertainty := 0;
    sDescription := 'Atomic mass of Co (cobalt)';
    sUnits := 'None';
    sCaveat := 'None';
    bFound := TRUE;
ELSIF sName = 'Ni' THEN
    fValue := 58.6934;
    fUncertainty := 0;
    sDescription := 'Atomic mass of Ni (nickel)';
    sUnits := 'None';
    sCaveat := 'None';
    bFound := TRUE;
ELSIF sName = 'Cu' THEN
    fValue := 63.546;
    fUncertainty := 0;
    sDescription := 'Atomic mass of Cu (copper)';
    sUnits := 'None';
    sCaveat := 'None';
    bFound := TRUE;
ELSIF sName = 'Zn' THEN
    fValue := 65.409;
    fUncertainty := 0;
    sDescription := 'Atomic mass of Zn (zinc)';
    sUnits := 'None';
    sCaveat := 'None';
    bFound := TRUE;
ELSIF sName = 'Ga' THEN
    fValue := 69.723;
    fUncertainty := 0;
    sDescription := 'Atomic mass of Ga (gallium)';
    sUnits := 'None';
    sCaveat := 'None';
    bFound := TRUE;
ELSIF sName = 'Ge' THEN
    fValue := 72.64;
    fUncertainty := 0;
    sDescription := 'Atomic mass of Ge (germanium)';
    sUnits := 'None';
    sCaveat := 'None';
    bFound := TRUE;
ELSIF sName = 'As' THEN
    fValue := 74.9216;
    fUncertainty := 0;
    sDescription := 'Atomic mass of As (arsenic)';
    sUnits := 'None';
    sCaveat := 'None';
    bFound := TRUE;
ELSIF sName = 'Se' THEN
    fValue := 78.96;
    fUncertainty := 0;
    sDescription := 'Atomic mass of Se (selenium)';
    sUnits := 'None';
    sCaveat := 'None';
    bFound := TRUE;
ELSIF sName = 'Br' THEN
    fValue := 79.904;
    fUncertainty := 0;
    sDescription := 'Atomic mass of Br (bromine)';
    sUnits := 'None';
    sCaveat := 'None';
    bFound := TRUE;
ELSIF sName = 'Kr' THEN
    fValue := 83.798;
    fUncertainty := 0;
    sDescription := 'Atomic mass of Kr (krypton)';
    sUnits := 'None';
    sCaveat := 'None';
    bFound := TRUE;
ELSIF sName = 'Rb' THEN
    fValue := 85.4678;
    fUncertainty := 0;
    sDescription := 'Atomic mass of Rb (rubidium)';
    sUnits := 'None';
    sCaveat := 'None';
    bFound := TRUE;
ELSIF sName = 'Sr' THEN
    fValue := 87.62;
    fUncertainty := 0;
    sDescription := 'Atomic mass of Sr (strontium)';
    sUnits := 'None';
    sCaveat := 'None';
    bFound := TRUE;
ELSIF sName = 'Y' THEN
    fValue := 88.90585;
    fUncertainty := 0;
    sDescription := 'Atomic mass of Y (yttrium)';
    sUnits := 'None';
    sCaveat := 'None';
    bFound := TRUE;
ELSIF sName = 'Zr' THEN
    fValue := 91.224;
    fUncertainty := 0;
    sDescription := 'Atomic mass of Zr (zirconium)';
    sUnits := 'None';
    sCaveat := 'None';
    bFound := TRUE;
ELSIF sName = 'Nb' THEN
    fValue := 92.90638;
    fUncertainty := 0;
    sDescription := 'Atomic mass of Nb (niobium)';
    sUnits := 'None';
    sCaveat := 'None';
    bFound := TRUE;
ELSIF sName = 'Mo' THEN
    fValue := 95.94;
    fUncertainty := 0;
    sDescription := 'Atomic mass of Mo (molybdenum)';
    sUnits := 'None';
    sCaveat := 'None';
    bFound := TRUE;
ELSIF sName = 'Tc' THEN
    fValue := 98;
    fUncertainty := 0;
    sDescription := 'Atomic mass of Tc (technetium)';
    sUnits := 'None';
    sCaveat := 'None';
    bFound := TRUE;
ELSIF sName = 'Ru' THEN
    fValue := 101.07;
    fUncertainty := 0;
    sDescription := 'Atomic mass of Ru (ruthenium)';
    sUnits := 'None';
    sCaveat := 'None';
    bFound := TRUE;
ELSIF sName = 'Rh' THEN
    fValue := 102.9055;
    fUncertainty := 0;
    sDescription := 'Atomic mass of Rh (rhodium)';
    sUnits := 'None';
    sCaveat := 'None';
    bFound := TRUE;
ELSIF sName = 'Pd' THEN
    fValue := 106.42;
    fUncertainty := 0;
    sDescription := 'Atomic mass of Pd (palladium)';
    sUnits := 'None';
    sCaveat := 'None';
    bFound := TRUE;
ELSIF sName = 'Ag' THEN
    fValue := 107.8682;
    fUncertainty := 0;
    sDescription := 'Atomic mass of Ag (silver)';
    sUnits := 'None';
    sCaveat := 'None';
    bFound := TRUE;
ELSIF sName = 'Cd' THEN
    fValue := 112.411;
    fUncertainty := 0;
    sDescription := 'Atomic mass of Cd (cadmium)';
    sUnits := 'None';
    sCaveat := 'None';
    bFound := TRUE;
ELSIF sName = 'In' THEN
    fValue := 114.818;
    fUncertainty := 0;
    sDescription := 'Atomic mass of In (indium)';
    sUnits := 'None';
    sCaveat := 'None';
    bFound := TRUE;
ELSIF sName = 'Sn' THEN
    fValue := 118.71;
    fUncertainty := 0;
    sDescription := 'Atomic mass of Sn (tin)';
    sUnits := 'None';
    sCaveat := 'None';
    bFound := TRUE;
ELSIF sName = 'Sb' THEN
    fValue := 121.76;
    fUncertainty := 0;
    sDescription := 'Atomic mass of Sb (antimony)';
    sUnits := 'None';
    sCaveat := 'None';
    bFound := TRUE;
ELSIF sName = 'Te' THEN
    fValue := 127.6;
    fUncertainty := 0;
    sDescription := 'Atomic mass of Te (tellurium)';
    sUnits := 'None';
    sCaveat := 'None';
    bFound := TRUE;
ELSIF sName = 'I' THEN
    fValue := 126.90447;
    fUncertainty := 0;
    sDescription := 'Atomic mass of I (iodine)';
    sUnits := 'None';
    sCaveat := 'None';
    bFound := TRUE;
ELSIF sName = 'Xe' THEN
    fValue := 131.293;
    fUncertainty := 0;
    sDescription := 'Atomic mass of Xe (xenon)';
    sUnits := 'None';
    sCaveat := 'None';
    bFound := TRUE;
ELSIF sName = 'Cs' THEN
    fValue := 132.90545;
    fUncertainty := 0;
    sDescription := 'Atomic mass of Cs (cesium)';
    sUnits := 'None';
    sCaveat := 'None';
    bFound := TRUE;
ELSIF sName = 'Ba' THEN
    fValue := 137.327;
    fUncertainty := 0;
    sDescription := 'Atomic mass of Ba (barium)';
    sUnits := 'None';
    sCaveat := 'None';
    bFound := TRUE;
ELSIF sName = 'La' THEN
    fValue := 138.9055;
    fUncertainty := 0;
    sDescription := 'Atomic mass of La (lanthanum)';
    sUnits := 'None';
    sCaveat := 'None';
    bFound := TRUE;
ELSIF sName = 'Ce' THEN
    fValue := 140.116;
    fUncertainty := 0;
    sDescription := 'Atomic mass of Ce (cerium)';
    sUnits := 'None';
    sCaveat := 'None';
    bFound := TRUE;
ELSIF sName = 'Pr' THEN
    fValue := 140.90765;
    fUncertainty := 0;
    sDescription := 'Atomic mass of Pr (praseodymium)';
    sUnits := 'None';
    sCaveat := 'None';
    bFound := TRUE;
ELSIF sName = 'Nd' THEN
    fValue := 144.24;
    fUncertainty := 0;
    sDescription := 'Atomic mass of Nd (neodymium)';
    sUnits := 'None';
    sCaveat := 'None';
    bFound := TRUE;
ELSIF sName = 'Pm' THEN
    fValue := 145;
    fUncertainty := 0;
    sDescription := 'Atomic mass of Pm (promethium)';
    sUnits := 'None';
    sCaveat := 'None';
    bFound := TRUE;
ELSIF sName = 'Sm' THEN
    fValue := 150.36;
    fUncertainty := 0;
    sDescription := 'Atomic mass of Sm (samarium)';
    sUnits := 'None';
    sCaveat := 'None';
    bFound := TRUE;
ELSIF sName = 'Eu' THEN
    fValue := 151.964;
    fUncertainty := 0;
    sDescription := 'Atomic mass of Eu (europium)';
    sUnits := 'None';
    sCaveat := 'None';
    bFound := TRUE;
ELSIF sName = 'Gd' THEN
    fValue := 157.25;
    fUncertainty := 0;
    sDescription := 'Atomic mass of Gd (gadolinium)';
    sUnits := 'None';
    sCaveat := 'None';
    bFound := TRUE;
ELSIF sName = 'Tb' THEN
    fValue := 158.92534;
    fUncertainty := 0;
    sDescription := 'Atomic mass of Tb (terbium)';
    sUnits := 'None';
    sCaveat := 'None';
    bFound := TRUE;
ELSIF sName = 'Dy' THEN
    fValue := 162.5;
    fUncertainty := 0;
    sDescription := 'Atomic mass of Dy (dysprosium)';
    sUnits := 'None';
    sCaveat := 'None';
    bFound := TRUE;
ELSIF sName = 'Ho' THEN
    fValue := 164.93032;
    fUncertainty := 0;
    sDescription := 'Atomic mass of Ho (holmium)';
    sUnits := 'None';
    sCaveat := 'None';
    bFound := TRUE;
ELSIF sName = 'Er' THEN
    fValue := 167.259;
    fUncertainty := 0;
    sDescription := 'Atomic mass of Er (erbium)';
    sUnits := 'None';
    sCaveat := 'None';
    bFound := TRUE;
ELSIF sName = 'Tm' THEN
    fValue := 168.93421;
    fUncertainty := 0;
    sDescription := 'Atomic mass of Tm (thulium)';
    sUnits := 'None';
    sCaveat := 'None';
    bFound := TRUE;
ELSIF sName = 'Yb' THEN
    fValue := 173.04;
    fUncertainty := 0;
    sDescription := 'Atomic mass of Yb (ytterbium)';
    sUnits := 'None';
    sCaveat := 'None';
    bFound := TRUE;
ELSIF sName = 'Lu' THEN
    fValue := 174.967;
    fUncertainty := 0;
    sDescription := 'Atomic mass of Lu (lutetium)';
    sUnits := 'None';
    sCaveat := 'None';
    bFound := TRUE;
ELSIF sName = 'Hf' THEN
    fValue := 178.49;
    fUncertainty := 0;
    sDescription := 'Atomic mass of Hf (hafnium)';
    sUnits := 'None';
    sCaveat := 'None';
    bFound := TRUE;
ELSIF sName = 'Ta' THEN
    fValue := 180.9479;
    fUncertainty := 0;
    sDescription := 'Atomic mass of Ta (tantalum)';
    sUnits := 'None';
    sCaveat := 'None';
    bFound := TRUE;
ELSIF sName = 'W' THEN
    fValue := 183.84;
    fUncertainty := 0;
    sDescription := 'Atomic mass of W (tungsten)';
    sUnits := 'None';
    sCaveat := 'None';
    bFound := TRUE;
ELSIF sName = 'Re' THEN
    fValue := 186.207;
    fUncertainty := 0;
    sDescription := 'Atomic mass of Re (rhenium)';
    sUnits := 'None';
    sCaveat := 'None';
    bFound := TRUE;
ELSIF sName = 'Os' THEN
    fValue := 190.23;
    fUncertainty := 0;
    sDescription := 'Atomic mass of Os (osmium)';
    sUnits := 'None';
    sCaveat := 'None';
    bFound := TRUE;
ELSIF sName = 'Ir' THEN
    fValue := 192.217;
    fUncertainty := 0;
    sDescription := 'Atomic mass of Ir (iridium)';
    sUnits := 'None';
    sCaveat := 'None';
    bFound := TRUE;
ELSIF sName = 'Pt' THEN
    fValue := 195.078;
    fUncertainty := 0;
    sDescription := 'Atomic mass of Pt (platinum)';
    sUnits := 'None';
    sCaveat := 'None';
    bFound := TRUE;
ELSIF sName = 'Au' THEN
    fValue := 196.96655;
    fUncertainty := 0;
    sDescription := 'Atomic mass of Au (gold)';
    sUnits := 'None';
    sCaveat := 'None';
    bFound := TRUE;
ELSIF sName = 'Hg' THEN
    fValue := 200.59;
    fUncertainty := 0;
    sDescription := 'Atomic mass of Hg (mercury)';
    sUnits := 'None';
    sCaveat := 'None';
    bFound := TRUE;
ELSIF sName = 'Tl' THEN
    fValue := 204.3833;
    fUncertainty := 0;
    sDescription := 'Atomic mass of Tl (thallium)';
    sUnits := 'None';
    sCaveat := 'None';
    bFound := TRUE;
ELSIF sName = 'Pb' THEN
    fValue := 207.2;
    fUncertainty := 0;
    sDescription := 'Atomic mass of Pb (lead)';
    sUnits := 'None';
    sCaveat := 'None';
    bFound := TRUE;
ELSIF sName = 'Bi' THEN
    fValue := 208.98038;
    fUncertainty := 0;
    sDescription := 'Atomic mass of Bi (bismuth)';
    sUnits := 'None';
    sCaveat := 'None';
    bFound := TRUE;
ELSIF sName = 'Po' THEN
    fValue := 209;
    fUncertainty := 0;
    sDescription := 'Atomic mass of Po (polonium)';
    sUnits := 'None';
    sCaveat := 'None';
    bFound := TRUE;
ELSIF sName = 'At' THEN
    fValue := 210;
    fUncertainty := 0;
    sDescription := 'Atomic mass of At (astatine)';
    sUnits := 'None';
    sCaveat := 'None';
    bFound := TRUE;
ELSIF sName = 'Rn' THEN
    fValue := 222;
    fUncertainty := 0;
    sDescription := 'Atomic mass of Rn (radon)';
    sUnits := 'None';
    sCaveat := 'None';
    bFound := TRUE;
ELSIF sName = 'Fr' THEN
    fValue := 223;
    fUncertainty := 0;
    sDescription := 'Atomic mass of Fr (francium)';
    sUnits := 'None';
    sCaveat := 'None';
    bFound := TRUE;
ELSIF sName = 'Ra' THEN
    fValue := 226;
    fUncertainty := 0;
    sDescription := 'Atomic mass of Ra (radium)';
    sUnits := 'None';
    sCaveat := 'None';
    bFound := TRUE;
ELSIF sName = 'Ac' THEN
    fValue := 227;
    fUncertainty := 0;
    sDescription := 'Atomic mass of Ac (actinium)';
    sUnits := 'None';
    sCaveat := 'None';
    bFound := TRUE;
ELSIF sName = 'Th' THEN
    fValue := 232.0381;
    fUncertainty := 0;
    sDescription := 'Atomic mass of Th (thorium)';
    sUnits := 'None';
    sCaveat := 'None';
    bFound := TRUE;
ELSIF sName = 'Pa' THEN
    fValue := 231.03588;
    fUncertainty := 0;
    sDescription := 'Atomic mass of Pa (protactinium)';
    sUnits := 'None';
    sCaveat := 'None';
    bFound := TRUE;
ELSIF sName = 'U' THEN
    fValue := 238.02891;
    fUncertainty := 0;
    sDescription := 'Atomic mass of U (uranium)';
    sUnits := 'None';
    sCaveat := 'None';
    bFound := TRUE;
ELSIF sName = 'Np' THEN
    fValue := 237;
    fUncertainty := 0;
    sDescription := 'Atomic mass of Np (neptunium)';
    sUnits := 'None';
    sCaveat := 'None';
    bFound := TRUE;
ELSIF sName = 'Pu' THEN
    fValue := 244;
    fUncertainty := 0;
    sDescription := 'Atomic mass of Pu (plutonium)';
    sUnits := 'None';
    sCaveat := 'None';
    bFound := TRUE;
ELSIF sName = 'Am' THEN
    fValue := 243;
    fUncertainty := 0;
    sDescription := 'Atomic mass of Am (americium)';
    sUnits := 'None';
    sCaveat := 'None';
    bFound := TRUE;
ELSIF sName = 'Cm' THEN
    fValue := 247;
    fUncertainty := 0;
    sDescription := 'Atomic mass of Cm (curium)';
    sUnits := 'None';
    sCaveat := 'None';
    bFound := TRUE;
ELSIF sName = 'Bk' THEN
    fValue := 247;
    fUncertainty := 0;
    sDescription := 'Atomic mass of Bk (berkelium)';
    sUnits := 'None';
    sCaveat := 'None';
    bFound := TRUE;
ELSIF sName = 'Cf' THEN
    fValue := 251;
    fUncertainty := 0;
    sDescription := 'Atomic mass of Cf (californium)';
    sUnits := 'None';
    sCaveat := 'None';
    bFound := TRUE;
ELSIF sName = 'Es' THEN
    fValue := 252;
    fUncertainty := 0;
    sDescription := 'Atomic mass of Es (einsteinium)';
    sUnits := 'None';
    sCaveat := 'None';
    bFound := TRUE;
ELSIF sName = 'Fm' THEN
    fValue := 257;
    fUncertainty := 0;
    sDescription := 'Atomic mass of Fm (fermium)';
    sUnits := 'None';
    sCaveat := 'None';
    bFound := TRUE;
ELSIF sName = 'Md' THEN
    fValue := 258;
    fUncertainty := 0;
    sDescription := 'Atomic mass of Md (mendelevium)';
    sUnits := 'None';
    sCaveat := 'None';
    bFound := TRUE;
ELSIF sName = 'No' THEN
    fValue := 259;
    fUncertainty := 0;
    sDescription := 'Atomic mass of No (nobelium)';
    sUnits := 'None';
    sCaveat := 'None';
    bFound := TRUE;
ELSIF sName = 'Lr' THEN
    fValue := 262;
    fUncertainty := 0;
    sDescription := 'Atomic mass of Lr (lawrencium)';
    sUnits := 'None';
    sCaveat := 'None';
    bFound := TRUE;
ELSIF sName = 'Rf' THEN
    fValue := 261;
    fUncertainty := 0;
    sDescription := 'Atomic mass of Rf (rutherfordium)';
    sUnits := 'None';
    sCaveat := 'None';
    bFound := TRUE;
ELSIF sName = 'Db' THEN
    fValue := 262;
    fUncertainty := 0;
    sDescription := 'Atomic mass of Db (dubnium)';
    sUnits := 'None';
    sCaveat := 'None';
    bFound := TRUE;
ELSIF sName = 'Sg' THEN
    fValue := 266;
    fUncertainty := 0;
    sDescription := 'Atomic mass of Sg (seaborgium)';
    sUnits := 'None';
    sCaveat := 'None';
    bFound := TRUE;
ELSIF sName = 'Bh' THEN
    fValue := 264;
    fUncertainty := 0;
    sDescription := 'Atomic mass of Bh (bohrium)';
    sUnits := 'None';
    sCaveat := 'None';
    bFound := TRUE;
ELSIF sName = 'Hs' THEN
    fValue := 277;
    fUncertainty := 0;
    sDescription := 'Atomic mass of Hs (hassium)';
    sUnits := 'None';
    sCaveat := 'None';
    bFound := TRUE;
ELSIF sName = 'Mt' THEN
    fValue := 268;
    fUncertainty := 0;
    sDescription := 'Atomic mass of Mt (meitnerium)';
    sUnits := 'None';
    sCaveat := 'None';
    bFound := TRUE;
ELSIF sName = 'Ds' THEN
    fValue := 281;
    fUncertainty := 0;
    sDescription := 'Atomic mass of Ds (darmstadtium)';
    sUnits := 'None';
    sCaveat := 'None';
    bFound := TRUE;
ELSIF sName = 'Rg' THEN
    fValue := 272;
    fUncertainty := 0;
    sDescription := 'Atomic mass of Rg (roentgenium)';
    sUnits := 'None';
    sCaveat := 'None';
    bFound := TRUE;
ELSIF sName = 'Cn' THEN
    fValue := 285;
    fUncertainty := 0;
    sDescription := 'Atomic mass of Cn (copernicium)';
    sUnits := 'None';
    sCaveat := 'None';
    bFound := TRUE;
ELSIF sName = 'Nh' THEN
    fValue := 286;
    fUncertainty := 0;
    sDescription := 'Atomic mass of Nh (nihonium)';
    sUnits := 'None';
    sCaveat := 'None';
    bFound := TRUE;
ELSIF sName = 'Fl' THEN
    fValue := 289;
    fUncertainty := 0;
    sDescription := 'Atomic mass of Fl (flerovium)';
    sUnits := 'None';
    sCaveat := 'None';
    bFound := TRUE;
ELSIF sName = 'Mc' THEN
    fValue := 289;
    fUncertainty := 0;
    sDescription := 'Atomic mass of Mc (moscovium)';
    sUnits := 'None';
    sCaveat := 'None';
    bFound := TRUE;
ELSIF sName = 'Lv' THEN
    fValue := 293;
    fUncertainty := 0;
    sDescription := 'Atomic mass of Lv (livermorium)';
    sUnits := 'None';
    sCaveat := 'None';
    bFound := TRUE;
ELSIF sName = 'Ts' THEN
    fValue := 294;
    fUncertainty := 0;
    sDescription := 'Atomic mass of Ts (tennessine)';
    sUnits := 'None';
    sCaveat := 'None';
    bFound := TRUE;
ELSIF sName = 'Og' THEN
    fValue := 294;
    fUncertainty := 0;
    sDescription := 'Atomic mass of Og (oganesson)';
    sUnits := 'None';
    sCaveat := 'None';
    bFound := TRUE;
ELSE
    bFound := FALSE;
    fValue := 0;
    fUncertainty := 0;
    sDescription := '';
    sUnits := '';
    sCaveat := '';
END_IF

END_FUNCTION_BLOCK

// ---- Tests/FB_AtomicNumberLookup_Test.TcPOU

FUNCTION_BLOCK FB_AtomicNumberLookup_Test EXTENDS TcUnit.FB_TestSuite
VAR
END_VAR


GivenElementExpectCorrectAtomicNumber();


METHOD PRIVATE GivenElementExpectCorrectAtomicNumber
VAR
    nResult : INT;
END_VAR

TEST('GivenElementExpectCorrectAtomicNumber');

nResult := F_AtomicNumberLookup(
    sMaterialName := 'C'
);

AssertEquals_INT(
    Expected := 6,
    Actual := nResult,
    Message := 'Incorrect result.'
);

nResult := F_AtomicNumberLookup(
    sMaterialName := 'Cu'
);

AssertEquals_INT(
    Expected := 29,
    Actual := nResult,
    Message := 'Incorrect result.'
);

nResult := F_AtomicNumberLookup(
    sMaterialName := 'Be'
);

AssertEquals_INT(
    Expected := 4,
    Actual := nResult,
    Message := 'Incorrect result.'
);

TEST_FINISHED();
END_METHOD

END_FUNCTION_BLOCK

// ---- POUs/F_AtomicNumberLookup.TcPOU

FUNCTION F_AtomicNumberLookup : INT
VAR_INPUT
    sMaterialName : T_MaxString;
END_VAR
VAR
    fbAtomicNumber : FB_AtomicNumber;
END_VAR


fbAtomicNumber(
    sName := sMaterialName
);

IF fbAtomicNumber.bFound THEN
    F_AtomicNumberLookup := fbAtomicNumber.nValue;
ELSE
    F_AtomicNumberLookup := -1;
END_IF

END_FUNCTION

// ---- POUs/FB_AtomicNumber.TcPOU

(* WARNING: This file is auto-generated. Do not modify it.*)
FUNCTION_BLOCK FB_AtomicNumber

VAR_INPUT
    sName : STRING;
END_VAR

VAR_OUTPUT
    bFound : BOOL;
    nValue : INT;
    fUncertainty : LREAL;
    sDescription : STRING;
    sUnits : STRING;
    sCaveat : STRING;
END_VAR


(* WARNING: This file is auto-generated. Do not modify it.*)
IF sName = 'n' THEN
    nValue := 0;
    fUncertainty := 0;
    sDescription := 'Atomic number of n (neutron)';
    sUnits := 'None';
    sCaveat := 'None';
    bFound := TRUE;
ELSIF sName = 'H' THEN
    nValue := 1;
    fUncertainty := 0;
    sDescription := 'Atomic number of H (hydrogen)';
    sUnits := 'None';
    sCaveat := 'None';
    bFound := TRUE;
ELSIF sName = 'He' THEN
    nValue := 2;
    fUncertainty := 0;
    sDescription := 'Atomic number of He (helium)';
    sUnits := 'None';
    sCaveat := 'None';
    bFound := TRUE;
ELSIF sName = 'Li' THEN
    nValue := 3;
    fUncertainty := 0;
    sDescription := 'Atomic number of Li (lithium)';
    sUnits := 'None';
    sCaveat := 'None';
    bFound := TRUE;
ELSIF sName = 'Be' THEN
    nValue := 4;
    fUncertainty := 0;
    sDescription := 'Atomic number of Be (beryllium)';
    sUnits := 'None';
    sCaveat := 'None';
    bFound := TRUE;
ELSIF sName = 'B' THEN
    nValue := 5;
    fUncertainty := 0;
    sDescription := 'Atomic number of B (boron)';
    sUnits := 'None';
    sCaveat := 'None';
    bFound := TRUE;
ELSIF sName = 'C' OR sName = 'C (Diamond)' THEN
    nValue := 6;
    fUncertainty := 0;
    sDescription := 'Atomic number of C (carbon)';
    sUnits := 'None';
    sCaveat := 'None';
    bFound := TRUE;
ELSIF sName = 'N' THEN
    nValue := 7;
    fUncertainty := 0;
    sDescription := 'Atomic number of N (nitrogen)';
    sUnits := 'None';
    sCaveat := 'None';
    bFound := TRUE;
ELSIF sName = 'O' THEN
    nValue := 8;
    fUncertainty := 0;
    sDescription := 'Atomic number of O (oxygen)';
    sUnits := 'None';
    sCaveat := 'None';
    bFound := TRUE;
ELSIF sName = 'F' THEN
    nValue := 9;
    fUncertainty := 0;
    sDescription := 'Atomic number of F (fluorine)';
    sUnits := 'None';
    sCaveat := 'None';
    bFound := TRUE;
ELSIF sName = 'Ne' THEN
    nValue := 10;
    fUncertainty := 0;
    sDescription := 'Atomic number of Ne (neon)';
    sUnits := 'None';
    sCaveat := 'None';
    bFound := TRUE;
ELSIF sName = 'Na' THEN
    nValue := 11;
    fUncertainty := 0;
    sDescription := 'Atomic number of Na (sodium)';
    sUnits := 'None';
    sCaveat := 'None';
    bFound := TRUE;
ELSIF sName = 'Mg' THEN
    nValue := 12;
    fUncertainty := 0;
    sDescription := 'Atomic number of Mg (magnesium)';
    sUnits := 'None';
    sCaveat := 'None';
    bFound := TRUE;
ELSIF sName = 'Al' THEN
    nValue := 13;
    fUncertainty := 0;
    sDescription := 'Atomic number of Al (aluminum)';
    sUnits := 'None';
    sCaveat := 'None';
    bFound := TRUE;
ELSIF sName = 'Si' THEN
    nValue := 14;
    fUncertainty := 0;
    sDescription := 'Atomic number of Si (silicon)';
    sUnits := 'None';
    sCaveat := 'None';
    bFound := TRUE;
ELSIF sName = 'P' THEN
    nValue := 15;
    fUncertainty := 0;
    sDescription := 'Atomic number of P (phosphorus)';
    sUnits := 'None';
    sCaveat := 'None';
    bFound := TRUE;
ELSIF sName = 'S' THEN
    nValue := 16;
    fUncertainty := 0;
    sDescription := 'Atomic number of S (sulfur)';
    sUnits := 'None';
    sCaveat := 'None';
    bFound := TRUE;
ELSIF sName = 'Cl' THEN
    nValue := 17;
    fUncertainty := 0;
    sDescription := 'Atomic number of Cl (chlorine)';
    sUnits := 'None';
    sCaveat := 'None';
    bFound := TRUE;
ELSIF sName = 'Ar' THEN
    nValue := 18;
    fUncertainty := 0;
    sDescription := 'Atomic number of Ar (argon)';
    sUnits := 'None';
    sCaveat := 'None';
    bFound := TRUE;
ELSIF sName = 'K' THEN
    nValue := 19;
    fUncertainty := 0;
    sDescription := 'Atomic number of K (potassium)';
    sUnits := 'None';
    sCaveat := 'None';
    bFound := TRUE;
ELSIF sName = 'Ca' THEN
    nValue := 20;
    fUncertainty := 0;
    sDescription := 'Atomic number of Ca (calcium)';
    sUnits := 'None';
    sCaveat := 'None';
    bFound := TRUE;
ELSIF sName = 'Sc' THEN
    nValue := 21;
    fUncertainty := 0;
    sDescription := 'Atomic number of Sc (scandium)';
    sUnits := 'None';
    sCaveat := 'None';
    bFound := TRUE;
ELSIF sName = 'Ti' THEN
    nValue := 22;
    fUncertainty := 0;
    sDescription := 'Atomic number of Ti (titanium)';
    sUnits := 'None';
    sCaveat := 'None';
    bFound := TRUE;
ELSIF sName = 'V' THEN
    nValue := 23;
    fUncertainty := 0;
    sDescription := 'Atomic number of V (vanadium)';
    sUnits := 'None';
    sCaveat := 'None';
    bFound := TRUE;
ELSIF sName = 'Cr' THEN
    nValue := 24;
    fUncertainty := 0;
    sDescription := 'Atomic number of Cr (chromium)';
    sUnits := 'None';
    sCaveat := 'None';
    bFound := TRUE;
ELSIF sName = 'Mn' THEN
    nValue := 25;
    fUncertainty := 0;
    sDescription := 'Atomic number of Mn (manganese)';
    sUnits := 'None';
    sCaveat := 'None';
    bFound := TRUE;
ELSIF sName = 'Fe' THEN
    nValue := 26;
    fUncertainty := 0;
    sDescription := 'Atomic number of Fe (iron)';
    sUnits := 'None';
    sCaveat := 'None';
    bFound := TRUE;
ELSIF sName = 'Co' THEN
    nValue := 27;
    fUncertainty := 0;
    sDescription := 'Atomic number of Co (cobalt)';
    sUnits := 'None';
    sCaveat := 'None';
    bFound := TRUE;
ELSIF sName = 'Ni' THEN
    nValue := 28;
    fUncertainty := 0;
    sDescription := 'Atomic number of Ni (nickel)';
    sUnits := 'None';
    sCaveat := 'None';
    bFound := TRUE;
ELSIF sName = 'Cu' THEN
    nValue := 29;
    fUncertainty := 0;
    sDescription := 'Atomic number of Cu (copper)';
    sUnits := 'None';
    sCaveat := 'None';
    bFound := TRUE;
ELSIF sName = 'Zn' THEN
    nValue := 30;
    fUncertainty := 0;
    sDescription := 'Atomic number of Zn (zinc)';
    sUnits := 'None';
    sCaveat := 'None';
    bFound := TRUE;
ELSIF sName = 'Ga' THEN
    nValue := 31;
    fUncertainty := 0;
    sDescription := 'Atomic number of Ga (gallium)';
    sUnits := 'None';
    sCaveat := 'None';
    bFound := TRUE;
ELSIF sName = 'Ge' THEN
    nValue := 32;
    fUncertainty := 0;
    sDescription := 'Atomic number of Ge (germanium)';
    sUnits := 'None';
    sCaveat := 'None';
    bFound := TRUE;
ELSIF sName = 'As' THEN
    nValue := 33;
    fUncertainty := 0;
    sDescription := 'Atomic number of As (arsenic)';
    sUnits := 'None';
    sCaveat := 'None';
    bFound := TRUE;
ELSIF sName = 'Se' THEN
    nValue := 34;
    fUncertainty := 0;
    sDescription := 'Atomic number of Se (selenium)';
    sUnits := 'None';
    sCaveat := 'None';
    bFound := TRUE;
ELSIF sName = 'Br' THEN
    nValue := 35;
    fUncertainty := 0;
    sDescription := 'Atomic number of Br (bromine)';
    sUnits := 'None';
    sCaveat := 'None';
    bFound := TRUE;
ELSIF sName = 'Kr' THEN
    nValue := 36;
    fUncertainty := 0;
    sDescription := 'Atomic number of Kr (krypton)';
    sUnits := 'None';
    sCaveat := 'None';
    bFound := TRUE;
ELSIF sName = 'Rb' THEN
    nValue := 37;
    fUncertainty := 0;
    sDescription := 'Atomic number of Rb (rubidium)';
    sUnits := 'None';
    sCaveat := 'None';
    bFound := TRUE;
ELSIF sName = 'Sr' THEN
    nValue := 38;
    fUncertainty := 0;
    sDescription := 'Atomic number of Sr (strontium)';
    sUnits := 'None';
    sCaveat := 'None';
    bFound := TRUE;
ELSIF sName = 'Y' THEN
    nValue := 39;
    fUncertainty := 0;
    sDescription := 'Atomic number of Y (yttrium)';
    sUnits := 'None';
    sCaveat := 'None';
    bFound := TRUE;
ELSIF sName = 'Zr' THEN
    nValue := 40;
    fUncertainty := 0;
    sDescription := 'Atomic number of Zr (zirconium)';
    sUnits := 'None';
    sCaveat := 'None';
    bFound := TRUE;
ELSIF sName = 'Nb' THEN
    nValue := 41;
    fUncertainty := 0;
    sDescription := 'Atomic number of Nb (niobium)';
    sUnits := 'None';
    sCaveat := 'None';
    bFound := TRUE;
ELSIF sName = 'Mo' THEN
    nValue := 42;
    fUncertainty := 0;
    sDescription := 'Atomic number of Mo (molybdenum)';
    sUnits := 'None';
    sCaveat := 'None';
    bFound := TRUE;
ELSIF sName = 'Tc' THEN
    nValue := 43;
    fUncertainty := 0;
    sDescription := 'Atomic number of Tc (technetium)';
    sUnits := 'None';
    sCaveat := 'None';
    bFound := TRUE;
ELSIF sName = 'Ru' THEN
    nValue := 44;
    fUncertainty := 0;
    sDescription := 'Atomic number of Ru (ruthenium)';
    sUnits := 'None';
    sCaveat := 'None';
    bFound := TRUE;
ELSIF sName = 'Rh' THEN
    nValue := 45;
    fUncertainty := 0;
    sDescription := 'Atomic number of Rh (rhodium)';
    sUnits := 'None';
    sCaveat := 'None';
    bFound := TRUE;
ELSIF sName = 'Pd' THEN
    nValue := 46;
    fUncertainty := 0;
    sDescription := 'Atomic number of Pd (palladium)';
    sUnits := 'None';
    sCaveat := 'None';
    bFound := TRUE;
ELSIF sName = 'Ag' THEN
    nValue := 47;
    fUncertainty := 0;
    sDescription := 'Atomic number of Ag (silver)';
    sUnits := 'None';
    sCaveat := 'None';
    bFound := TRUE;
ELSIF sName = 'Cd' THEN
    nValue := 48;
    fUncertainty := 0;
    sDescription := 'Atomic number of Cd (cadmium)';
    sUnits := 'None';
    sCaveat := 'None';
    bFound := TRUE;
ELSIF sName = 'In' THEN
    nValue := 49;
    fUncertainty := 0;
    sDescription := 'Atomic number of In (indium)';
    sUnits := 'None';
    sCaveat := 'None';
    bFound := TRUE;
ELSIF sName = 'Sn' THEN
    nValue := 50;
    fUncertainty := 0;
    sDescription := 'Atomic number of Sn (tin)';
    sUnits := 'None';
    sCaveat := 'None';
    bFound := TRUE;
ELSIF sName = 'Sb' THEN
    nValue := 51;
    fUncertainty := 0;
    sDescription := 'Atomic number of Sb (antimony)';
    sUnits := 'None';
    sCaveat := 'None';
    bFound := TRUE;
ELSIF sName = 'Te' THEN
    nValue := 52;
    fUncertainty := 0;
    sDescription := 'Atomic number of Te (tellurium)';
    sUnits := 'None';
    sCaveat := 'None';
    bFound := TRUE;
ELSIF sName = 'I' THEN
    nValue := 53;
    fUncertainty := 0;
    sDescription := 'Atomic number of I (iodine)';
    sUnits := 'None';
    sCaveat := 'None';
    bFound := TRUE;
ELSIF sName = 'Xe' THEN
    nValue := 54;
    fUncertainty := 0;
    sDescription := 'Atomic number of Xe (xenon)';
    sUnits := 'None';
    sCaveat := 'None';
    bFound := TRUE;
ELSIF sName = 'Cs' THEN
    nValue := 55;
    fUncertainty := 0;
    sDescription := 'Atomic number of Cs (cesium)';
    sUnits := 'None';
    sCaveat := 'None';
    bFound := TRUE;
ELSIF sName = 'Ba' THEN
    nValue := 56;
    fUncertainty := 0;
    sDescription := 'Atomic number of Ba (barium)';
    sUnits := 'None';
    sCaveat := 'None';
    bFound := TRUE;
ELSIF sName = 'La' THEN
    nValue := 57;
    fUncertainty := 0;
    sDescription := 'Atomic number of La (lanthanum)';
    sUnits := 'None';
    sCaveat := 'None';
    bFound := TRUE;
ELSIF sName = 'Ce' THEN
    nValue := 58;
    fUncertainty := 0;
    sDescription := 'Atomic number of Ce (cerium)';
    sUnits := 'None';
    sCaveat := 'None';
    bFound := TRUE;
ELSIF sName = 'Pr' THEN
    nValue := 59;
    fUncertainty := 0;
    sDescription := 'Atomic number of Pr (praseodymium)';
    sUnits := 'None';
    sCaveat := 'None';
    bFound := TRUE;
ELSIF sName = 'Nd' THEN
    nValue := 60;
    fUncertainty := 0;
    sDescription := 'Atomic number of Nd (neodymium)';
    sUnits := 'None';
    sCaveat := 'None';
    bFound := TRUE;
ELSIF sName = 'Pm' THEN
    nValue := 61;
    fUncertainty := 0;
    sDescription := 'Atomic number of Pm (promethium)';
    sUnits := 'None';
    sCaveat := 'None';
    bFound := TRUE;
ELSIF sName = 'Sm' THEN
    nValue := 62;
    fUncertainty := 0;
    sDescription := 'Atomic number of Sm (samarium)';
    sUnits := 'None';
    sCaveat := 'None';
    bFound := TRUE;
ELSIF sName = 'Eu' THEN
    nValue := 63;
    fUncertainty := 0;
    sDescription := 'Atomic number of Eu (europium)';
    sUnits := 'None';
    sCaveat := 'None';
    bFound := TRUE;
ELSIF sName = 'Gd' THEN
    nValue := 64;
    fUncertainty := 0;
    sDescription := 'Atomic number of Gd (gadolinium)';
    sUnits := 'None';
    sCaveat := 'None';
    bFound := TRUE;
ELSIF sName = 'Tb' THEN
    nValue := 65;
    fUncertainty := 0;
    sDescription := 'Atomic number of Tb (terbium)';
    sUnits := 'None';
    sCaveat := 'None';
    bFound := TRUE;
ELSIF sName = 'Dy' THEN
    nValue := 66;
    fUncertainty := 0;
    sDescription := 'Atomic number of Dy (dysprosium)';
    sUnits := 'None';
    sCaveat := 'None';
    bFound := TRUE;
ELSIF sName = 'Ho' THEN
    nValue := 67;
    fUncertainty := 0;
    sDescription := 'Atomic number of Ho (holmium)';
    sUnits := 'None';
    sCaveat := 'None';
    bFound := TRUE;
ELSIF sName = 'Er' THEN
    nValue := 68;
    fUncertainty := 0;
    sDescription := 'Atomic number of Er (erbium)';
    sUnits := 'None';
    sCaveat := 'None';
    bFound := TRUE;
ELSIF sName = 'Tm' THEN
    nValue := 69;
    fUncertainty := 0;
    sDescription := 'Atomic number of Tm (thulium)';
    sUnits := 'None';
    sCaveat := 'None';
    bFound := TRUE;
ELSIF sName = 'Yb' THEN
    nValue := 70;
    fUncertainty := 0;
    sDescription := 'Atomic number of Yb (ytterbium)';
    sUnits := 'None';
    sCaveat := 'None';
    bFound := TRUE;
ELSIF sName = 'Lu' THEN
    nValue := 71;
    fUncertainty := 0;
    sDescription := 'Atomic number of Lu (lutetium)';
    sUnits := 'None';
    sCaveat := 'None';
    bFound := TRUE;
ELSIF sName = 'Hf' THEN
    nValue := 72;
    fUncertainty := 0;
    sDescription := 'Atomic number of Hf (hafnium)';
    sUnits := 'None';
    sCaveat := 'None';
    bFound := TRUE;
ELSIF sName = 'Ta' THEN
    nValue := 73;
    fUncertainty := 0;
    sDescription := 'Atomic number of Ta (tantalum)';
    sUnits := 'None';
    sCaveat := 'None';
    bFound := TRUE;
ELSIF sName = 'W' THEN
    nValue := 74;
    fUncertainty := 0;
    sDescription := 'Atomic number of W (tungsten)';
    sUnits := 'None';
    sCaveat := 'None';
    bFound := TRUE;
ELSIF sName = 'Re' THEN
    nValue := 75;
    fUncertainty := 0;
    sDescription := 'Atomic number of Re (rhenium)';
    sUnits := 'None';
    sCaveat := 'None';
    bFound := TRUE;
ELSIF sName = 'Os' THEN
    nValue := 76;
    fUncertainty := 0;
    sDescription := 'Atomic number of Os (osmium)';
    sUnits := 'None';
    sCaveat := 'None';
    bFound := TRUE;
ELSIF sName = 'Ir' THEN
    nValue := 77;
    fUncertainty := 0;
    sDescription := 'Atomic number of Ir (iridium)';
    sUnits := 'None';
    sCaveat := 'None';
    bFound := TRUE;
ELSIF sName = 'Pt' THEN
    nValue := 78;
    fUncertainty := 0;
    sDescription := 'Atomic number of Pt (platinum)';
    sUnits := 'None';
    sCaveat := 'None';
    bFound := TRUE;
ELSIF sName = 'Au' THEN
    nValue := 79;
    fUncertainty := 0;
    sDescription := 'Atomic number of Au (gold)';
    sUnits := 'None';
    sCaveat := 'None';
    bFound := TRUE;
ELSIF sName = 'Hg' THEN
    nValue := 80;
    fUncertainty := 0;
    sDescription := 'Atomic number of Hg (mercury)';
    sUnits := 'None';
    sCaveat := 'None';
    bFound := TRUE;
ELSIF sName = 'Tl' THEN
    nValue := 81;
    fUncertainty := 0;
    sDescription := 'Atomic number of Tl (thallium)';
    sUnits := 'None';
    sCaveat := 'None';
    bFound := TRUE;
ELSIF sName = 'Pb' THEN
    nValue := 82;
    fUncertainty := 0;
    sDescription := 'Atomic number of Pb (lead)';
    sUnits := 'None';
    sCaveat := 'None';
    bFound := TRUE;
ELSIF sName = 'Bi' THEN
    nValue := 83;
    fUncertainty := 0;
    sDescription := 'Atomic number of Bi (bismuth)';
    sUnits := 'None';
    sCaveat := 'None';
    bFound := TRUE;
ELSIF sName = 'Po' THEN
    nValue := 84;
    fUncertainty := 0;
    sDescription := 'Atomic number of Po (polonium)';
    sUnits := 'None';
    sCaveat := 'None';
    bFound := TRUE;
ELSIF sName = 'At' THEN
    nValue := 85;
    fUncertainty := 0;
    sDescription := 'Atomic number of At (astatine)';
    sUnits := 'None';
    sCaveat := 'None';
    bFound := TRUE;
ELSIF sName = 'Rn' THEN
    nValue := 86;
    fUncertainty := 0;
    sDescription := 'Atomic number of Rn (radon)';
    sUnits := 'None';
    sCaveat := 'None';
    bFound := TRUE;
ELSIF sName = 'Fr' THEN
    nValue := 87;
    fUncertainty := 0;
    sDescription := 'Atomic number of Fr (francium)';
    sUnits := 'None';
    sCaveat := 'None';
    bFound := TRUE;
ELSIF sName = 'Ra' THEN
    nValue := 88;
    fUncertainty := 0;
    sDescription := 'Atomic number of Ra (radium)';
    sUnits := 'None';
    sCaveat := 'None';
    bFound := TRUE;
ELSIF sName = 'Ac' THEN
    nValue := 89;
    fUncertainty := 0;
    sDescription := 'Atomic number of Ac (actinium)';
    sUnits := 'None';
    sCaveat := 'None';
    bFound := TRUE;
ELSIF sName = 'Th' THEN
    nValue := 90;
    fUncertainty := 0;
    sDescription := 'Atomic number of Th (thorium)';
    sUnits := 'None';
    sCaveat := 'None';
    bFound := TRUE;
ELSIF sName = 'Pa' THEN
    nValue := 91;
    fUncertainty := 0;
    sDescription := 'Atomic number of Pa (protactinium)';
    sUnits := 'None';
    sCaveat := 'None';
    bFound := TRUE;
ELSIF sName = 'U' THEN
    nValue := 92;
    fUncertainty := 0;
    sDescription := 'Atomic number of U (uranium)';
    sUnits := 'None';
    sCaveat := 'None';
    bFound := TRUE;
ELSIF sName = 'Np' THEN
    nValue := 93;
    fUncertainty := 0;
    sDescription := 'Atomic number of Np (neptunium)';
    sUnits := 'None';
    sCaveat := 'None';
    bFound := TRUE;
ELSIF sName = 'Pu' THEN
    nValue := 94;
    fUncertainty := 0;
    sDescription := 'Atomic number of Pu (plutonium)';
    sUnits := 'None';
    sCaveat := 'None';
    bFound := TRUE;
ELSIF sName = 'Am' THEN
    nValue := 95;
    fUncertainty := 0;
    sDescription := 'Atomic number of Am (americium)';
    sUnits := 'None';
    sCaveat := 'None';
    bFound := TRUE;
ELSIF sName = 'Cm' THEN
    nValue := 96;
    fUncertainty := 0;
    sDescription := 'Atomic number of Cm (curium)';
    sUnits := 'None';
    sCaveat := 'None';
    bFound := TRUE;
ELSIF sName = 'Bk' THEN
    nValue := 97;
    fUncertainty := 0;
    sDescription := 'Atomic number of Bk (berkelium)';
    sUnits := 'None';
    sCaveat := 'None';
    bFound := TRUE;
ELSIF sName = 'Cf' THEN
    nValue := 98;
    fUncertainty := 0;
    sDescription := 'Atomic number of Cf (californium)';
    sUnits := 'None';
    sCaveat := 'None';
    bFound := TRUE;
ELSIF sName = 'Es' THEN
    nValue := 99;
    fUncertainty := 0;
    sDescription := 'Atomic number of Es (einsteinium)';
    sUnits := 'None';
    sCaveat := 'None';
    bFound := TRUE;
ELSIF sName = 'Fm' THEN
    nValue := 100;
    fUncertainty := 0;
    sDescription := 'Atomic number of Fm (fermium)';
    sUnits := 'None';
    sCaveat := 'None';
    bFound := TRUE;
ELSIF sName = 'Md' THEN
    nValue := 101;
    fUncertainty := 0;
    sDescription := 'Atomic number of Md (mendelevium)';
    sUnits := 'None';
    sCaveat := 'None';
    bFound := TRUE;
ELSIF sName = 'No' THEN
    nValue := 102;
    fUncertainty := 0;
    sDescription := 'Atomic number of No (nobelium)';
    sUnits := 'None';
    sCaveat := 'None';
    bFound := TRUE;
ELSIF sName = 'Lr' THEN
    nValue := 103;
    fUncertainty := 0;
    sDescription := 'Atomic number of Lr (lawrencium)';
    sUnits := 'None';
    sCaveat := 'None';
    bFound := TRUE;
ELSIF sName = 'Rf' THEN
    nValue := 104;
    fUncertainty := 0;
    sDescription := 'Atomic number of Rf (rutherfordium)';
    sUnits := 'None';
    sCaveat := 'None';
    bFound := TRUE;
ELSIF sName = 'Db' THEN
    nValue := 105;
    fUncertainty := 0;
    sDescription := 'Atomic number of Db (dubnium)';
    sUnits := 'None';
    sCaveat := 'None';
    bFound := TRUE;
ELSIF sName = 'Sg' THEN
    nValue := 106;
    fUncertainty := 0;
    sDescription := 'Atomic number of Sg (seaborgium)';
    sUnits := 'None';
    sCaveat := 'None';
    bFound := TRUE;
ELSIF sName = 'Bh' THEN
    nValue := 107;
    fUncertainty := 0;
    sDescription := 'Atomic number of Bh (bohrium)';
    sUnits := 'None';
    sCaveat := 'None';
    bFound := TRUE;
ELSIF sName = 'Hs' THEN
    nValue := 108;
    fUncertainty := 0;
    sDescription := 'Atomic number of Hs (hassium)';
    sUnits := 'None';
    sCaveat := 'None';
    bFound := TRUE;
ELSIF sName = 'Mt' THEN
    nValue := 109;
    fUncertainty := 0;
    sDescription := 'Atomic number of Mt (meitnerium)';
    sUnits := 'None';
    sCaveat := 'None';
    bFound := TRUE;
ELSIF sName = 'Ds' THEN
    nValue := 110;
    fUncertainty := 0;
    sDescription := 'Atomic number of Ds (darmstadtium)';
    sUnits := 'None';
    sCaveat := 'None';
    bFound := TRUE;
ELSIF sName = 'Rg' THEN
    nValue := 111;
    fUncertainty := 0;
    sDescription := 'Atomic number of Rg (roentgenium)';
    sUnits := 'None';
    sCaveat := 'None';
    bFound := TRUE;
ELSIF sName = 'Cn' THEN
    nValue := 112;
    fUncertainty := 0;
    sDescription := 'Atomic number of Cn (copernicium)';
    sUnits := 'None';
    sCaveat := 'None';
    bFound := TRUE;
ELSIF sName = 'Nh' THEN
    nValue := 113;
    fUncertainty := 0;
    sDescription := 'Atomic number of Nh (nihonium)';
    sUnits := 'None';
    sCaveat := 'None';
    bFound := TRUE;
ELSIF sName = 'Fl' THEN
    nValue := 114;
    fUncertainty := 0;
    sDescription := 'Atomic number of Fl (flerovium)';
    sUnits := 'None';
    sCaveat := 'None';
    bFound := TRUE;
ELSIF sName = 'Mc' THEN
    nValue := 115;
    fUncertainty := 0;
    sDescription := 'Atomic number of Mc (moscovium)';
    sUnits := 'None';
    sCaveat := 'None';
    bFound := TRUE;
ELSIF sName = 'Lv' THEN
    nValue := 116;
    fUncertainty := 0;
    sDescription := 'Atomic number of Lv (livermorium)';
    sUnits := 'None';
    sCaveat := 'None';
    bFound := TRUE;
ELSIF sName = 'Ts' THEN
    nValue := 117;
    fUncertainty := 0;
    sDescription := 'Atomic number of Ts (tennessine)';
    sUnits := 'None';
    sCaveat := 'None';
    bFound := TRUE;
ELSIF sName = 'Og' THEN
    nValue := 118;
    fUncertainty := 0;
    sDescription := 'Atomic number of Og (oganesson)';
    sUnits := 'None';
    sCaveat := 'None';
    bFound := TRUE;
ELSE
    bFound := FALSE;
    nValue := -1;
    fUncertainty := 0;
    sDescription := '';
    sUnits := '';
    sCaveat := '';
END_IF

END_FUNCTION_BLOCK

// ---- Tests/FB_CalculateXrayAbsorptionConstant_Test.TcPOU

FUNCTION_BLOCK FB_CalculateXrayAbsorptionConstant_Test EXTENDS TcUnit.FB_TestSuite
VAR
END_VAR


GivenValidInputsExpectCorrectResult();


METHOD PRIVATE GivenValidInputsExpectCorrectResult
VAR
    fResult : LREAL;
END_VAR

TEST('GivenValidInputsExpectCorrectResult');

fResult := F_CalculateXrayAbsorptionConstant(
    f2 := 0.0058932368755846573,
    fPhotonEnergy_eV := 10000,
    fDensity_gm3 := 3.51e6,
    fAtomicWeight := 12.0107
);

AssertEquals_LREAL(
    Expected := 724.7224642932565,
    Actual := fResult,
    Delta := 1e-9,
    Message := 'Incorrect result.'
);

TEST_FINISHED();
END_METHOD

END_FUNCTION_BLOCK

// ---- POUs/F_CalculateXrayAbsorptionConstant.TcPOU

FUNCTION F_CalculateXrayAbsorptionConstant : LREAL
(*
    Performs the same function as F_CalculateAbsorptionConstant, but
    the implementation has been decoupled from the particular lookup
    table used. New function made to retain backwards compatability.
    "F_CalculateXrayAbsorptionConstant" name used in order to make the new
    function distinguishable from the old one.
*)
VAR CONSTANT
    NA : LREAL := GVL_PhysicalConstants.fAvogadroConstant_in_mol_1;
    r0 : LREAL := GVL_PhysicalConstants.fClassicalElectronRadius_in_m;
    h  : LREAL := GVL_PhysicalConstants.fPlanckConstantInEV_Hz_in_eV_Hz_1;
    c  : LREAL := GVL_PhysicalConstants.fSpeedOfLightInVacuum_in_m_s_1;
END_VAR
VAR_INPUT
    f2 : LREAL; (* Scattering factor absorptive component. *)
    fPhotonEnergy_eV : LREAL;
    fDensity_gm3 : LREAL;
    fAtomicWeight : LREAL;
END_VAR


F_CalculateXrayAbsorptionConstant := (2.0 * r0 * h * c * f2 / fPhotonEnergy_eV) * fDensity_gm3 * (NA / fAtomicWeight);

END_FUNCTION

// ---- Tests/FB_CalculateThicknessFromTransmission_Test.TcPOU

FUNCTION_BLOCK FB_CalculateThicknessFromTransmission_Test EXTENDS TcUnit.FB_TestSuite
VAR
END_VAR


GivenTransmissionExpectCorrectThickness();


METHOD PRIVATE GivenTransmissionExpectCorrectThickness
VAR
    fResult : LREAL;
END_VAR

TEST('GivenTransmissionExpectCorrectThickness');

fResult := F_CalculateThicknessFromTransmission(
    fAbsorptionConstant := 724.7224642932565,
    fTransmission := 0.48445900560318955
);

AssertEquals_LREAL(
    Expected := 1e-3,
    Actual := fResult,
    Delta := 1e-9,
    Message := 'Incorrect result.'
);

TEST_FINISHED();
END_METHOD

END_FUNCTION_BLOCK

// ---- POUs/F_CalculateThicknessFromTransmission.TcPOU

FUNCTION F_CalculateThicknessFromTransmission : LREAL
(*
    Thickness returned in units of meters.
    Negative result means invalid input.
    Absorption constant must be greater than 0.
    Transmission must be between 0.0 and 1.0 inclusive.
*)
VAR_INPUT
    fAbsorptionConstant : LREAL; (* The absorption constant mu, calculated by F_CalculateXrayAbsorptionConstant *)
    fTransmission : LREAL; (* Transmission to get thickness for [unitless] *)
END_VAR


IF fAbsorptionConstant <= 0 OR fTransmission < 0.0 OR fTransmission > 1.0 THEN
    F_CalculateThicknessFromTransmission := -1.0;
    RETURN;
END_IF

F_CalculateThicknessFromTransmission := LN(fTransmission) / -fAbsorptionConstant;

END_FUNCTION

// ---- Tests/FB_MaterialDensityLookup_Test.TcPOU

FUNCTION_BLOCK FB_MaterialDensityLookup_Test EXTENDS TcUnit.FB_TestSuite
VAR
END_VAR


GivenElementExpectCorrectDensity();


METHOD PRIVATE GivenElementExpectCorrectDensity
VAR
    fResult : LREAL;
END_VAR

TEST('GivenElementExpectCorrectDensity');

fResult := F_MaterialDensityLookup(
    sMaterialName := 'C (Diamond)'
);

AssertEquals_LREAL(
    Expected := 3.51,
    Actual := fResult,
    Delta := 1e-9,
    Message := 'Incorrect result.'
);

TEST_FINISHED();
END_METHOD

END_FUNCTION_BLOCK

// ---- POUs/F_MaterialDensityLookup.TcPOU

FUNCTION F_MaterialDensityLookup : LREAL
VAR_INPUT
    sMaterialName : T_MaxString;
END_VAR
VAR
    fbElementDensity : FB_ElementDensity;
END_VAR


fbElementDensity(
    sName := sMaterialName
);

IF fbElementDensity.bFound THEN
    F_MaterialDensityLookup := fbElementDensity.fValue;
ELSE
    F_MaterialDensityLookup := -1.0;
END_IF

END_FUNCTION

// ---- POUs/FB_ElementDensity.TcPOU

(* WARNING: This file is auto-generated. Do not modify it.*)
FUNCTION_BLOCK FB_ElementDensity

VAR_INPUT
    sName : STRING;
END_VAR

VAR_OUTPUT
    bFound : BOOL;
    fValue : LREAL;
    fUncertainty : LREAL;
    sDescription : STRING;
    sUnits : STRING;
    sCaveat : STRING;
END_VAR


(* WARNING: This file is auto-generated. Do not modify it.*)
IF sName = 'H' THEN
    fValue := 0.0708; (* Units: g/cm^3 *)
    fUncertainty := 0;
    sDescription := 'Elemental density of H';
    sUnits := 'g/cm^3';
    sCaveat := 'T=-252.87';
    bFound := TRUE;
ELSIF sName = 'He' THEN
    fValue := 0.122; (* Units: g/cm^3 *)
    fUncertainty := 0;
    sDescription := 'Elemental density of He';
    sUnits := 'g/cm^3';
    sCaveat := 'T=-268.93';
    bFound := TRUE;
ELSIF sName = 'Li' THEN
    fValue := 0.534; (* Units: g/cm^3 *)
    fUncertainty := 0;
    sDescription := 'Elemental density of Li';
    sUnits := 'g/cm^3';
    sCaveat := '';
    bFound := TRUE;
ELSIF sName = 'Be' THEN
    fValue := 1.848; (* Units: g/cm^3 *)
    fUncertainty := 0;
    sDescription := 'Elemental density of Be';
    sUnits := 'g/cm^3';
    sCaveat := '';
    bFound := TRUE;
ELSIF sName = 'B' THEN
    fValue := 2.34; (* Units: g/cm^3 *)
    fUncertainty := 0;
    sDescription := 'Elemental density of B';
    sUnits := 'g/cm^3';
    sCaveat := '';
    bFound := TRUE;
ELSIF sName = 'C' THEN
    fValue := 2.2; (* Units: g/cm^3 *)
    fUncertainty := 0;
    sDescription := 'Elemental density of C';
    sUnits := 'g/cm^3';
    sCaveat := '1.9-2.3 (graphite); CXRO, RSC and CRC use 2.2; NIST Xray tables use 2.26';
    bFound := TRUE;
ELSIF sName = 'C (Diamond)' THEN
    fValue := 3.51; (* Units: g/cm^3 *)
    fUncertainty := 0;
    sDescription := 'Elemental density of diamond';
    sUnits := 'g/cm^3';
    sCaveat := '';
    bFound := TRUE;
ELSIF sName = 'N' THEN
    fValue := 0.808; (* Units: g/cm^3 *)
    fUncertainty := 0;
    sDescription := 'Elemental density of N';
    sUnits := 'g/cm^3';
    sCaveat := 'T=-195.79';
    bFound := TRUE;
ELSIF sName = 'O' THEN
    fValue := 1.14; (* Units: g/cm^3 *)
    fUncertainty := 0;
    sDescription := 'Elemental density of O';
    sUnits := 'g/cm^3';
    sCaveat := 'T=-182.95';
    bFound := TRUE;
ELSIF sName = 'F' THEN
    fValue := 1.5; (* Units: g/cm^3 *)
    fUncertainty := 0;
    sDescription := 'Elemental density of F';
    sUnits := 'g/cm^3';
    sCaveat := 'T=-188.12';
    bFound := TRUE;
ELSIF sName = 'Ne' THEN
    fValue := 1.207; (* Units: g/cm^3 *)
    fUncertainty := 0;
    sDescription := 'Elemental density of Ne';
    sUnits := 'g/cm^3';
    sCaveat := 'T=-246.08';
    bFound := TRUE;
ELSIF sName = 'Na' THEN
    fValue := 0.971; (* Units: g/cm^3 *)
    fUncertainty := 0;
    sDescription := 'Elemental density of Na';
    sUnits := 'g/cm^3';
    sCaveat := '';
    bFound := TRUE;
ELSIF sName = 'Mg' THEN
    fValue := 1.738; (* Units: g/cm^3 *)
    fUncertainty := 0;
    sDescription := 'Elemental density of Mg';
    sUnits := 'g/cm^3';
    sCaveat := '';
    bFound := TRUE;
ELSIF sName = 'Al' THEN
    fValue := 2.6989; (* Units: g/cm^3 *)
    fUncertainty := 0;
    sDescription := 'Elemental density of Al';
    sUnits := 'g/cm^3';
    sCaveat := '';
    bFound := TRUE;
ELSIF sName = 'Si' THEN
    fValue := 2.33; (* Units: g/cm^3 *)
    fUncertainty := 0;
    sDescription := 'Elemental density of Si';
    sUnits := 'g/cm^3';
    sCaveat := 'T=25';
    bFound := TRUE;
ELSIF sName = 'P' THEN
    fValue := 1.82; (* Units: g/cm^3 *)
    fUncertainty := 0;
    sDescription := 'Elemental density of P';
    sUnits := 'g/cm^3';
    sCaveat := '';
    bFound := TRUE;
ELSIF sName = 'S' THEN
    fValue := 2.07; (* Units: g/cm^3 *)
    fUncertainty := 0;
    sDescription := 'Elemental density of S';
    sUnits := 'g/cm^3';
    sCaveat := '';
    bFound := TRUE;
ELSIF sName = 'Cl' THEN
    fValue := 1.56; (* Units: g/cm^3 *)
    fUncertainty := 0;
    sDescription := 'Elemental density of Cl';
    sUnits := 'g/cm^3';
    sCaveat := 'T=-33.6, 0.44 C above boiling point';
    bFound := TRUE;
ELSIF sName = 'Ar' THEN
    fValue := 1.4; (* Units: g/cm^3 *)
    fUncertainty := 0;
    sDescription := 'Elemental density of Ar';
    sUnits := 'g/cm^3';
    sCaveat := 'T=-185.85';
    bFound := TRUE;
ELSIF sName = 'K' THEN
    fValue := 0.862; (* Units: g/cm^3 *)
    fUncertainty := 0;
    sDescription := 'Elemental density of K';
    sUnits := 'g/cm^3';
    sCaveat := '';
    bFound := TRUE;
ELSIF sName = 'Ca' THEN
    fValue := 1.55; (* Units: g/cm^3 *)
    fUncertainty := 0;
    sDescription := 'Elemental density of Ca';
    sUnits := 'g/cm^3';
    sCaveat := '';
    bFound := TRUE;
ELSIF sName = 'Sc' THEN
    fValue := 2.989; (* Units: g/cm^3 *)
    fUncertainty := 0;
    sDescription := 'Elemental density of Sc';
    sUnits := 'g/cm^3';
    sCaveat := 'T=25';
    bFound := TRUE;
ELSIF sName = 'Ti' THEN
    fValue := 4.54; (* Units: g/cm^3 *)
    fUncertainty := 0;
    sDescription := 'Elemental density of Ti';
    sUnits := 'g/cm^3';
    sCaveat := '';
    bFound := TRUE;
ELSIF sName = 'V' THEN
    fValue := 6.11; (* Units: g/cm^3 *)
    fUncertainty := 0;
    sDescription := 'Elemental density of V';
    sUnits := 'g/cm^3';
    sCaveat := 'T=18.7';
    bFound := TRUE;
ELSIF sName = 'Cr' THEN
    fValue := 7.19; (* Units: g/cm^3 *)
    fUncertainty := 0;
    sDescription := 'Elemental density of Cr';
    sUnits := 'g/cm^3';
    sCaveat := '7.18-7.20';
    bFound := TRUE;
ELSIF sName = 'Mn' THEN
    fValue := 7.33; (* Units: g/cm^3 *)
    fUncertainty := 0;
    sDescription := 'Elemental density of Mn';
    sUnits := 'g/cm^3';
    sCaveat := '7.21-7.44';
    bFound := TRUE;
ELSIF sName = 'Fe' THEN
    fValue := 7.874; (* Units: g/cm^3 *)
    fUncertainty := 0;
    sDescription := 'Elemental density of Fe';
    sUnits := 'g/cm^3';
    sCaveat := '';
    bFound := TRUE;
ELSIF sName = 'Co' THEN
    fValue := 8.9; (* Units: g/cm^3 *)
    fUncertainty := 0;
    sDescription := 'Elemental density of Co';
    sUnits := 'g/cm^3';
    sCaveat := '';
    bFound := TRUE;
ELSIF sName = 'Ni' THEN
    fValue := 8.902; (* Units: g/cm^3 *)
    fUncertainty := 0;
    sDescription := 'Elemental density of Ni';
    sUnits := 'g/cm^3';
    sCaveat := 'T=25';
    bFound := TRUE;
ELSIF sName = 'Cu' THEN
    fValue := 8.96; (* Units: g/cm^3 *)
    fUncertainty := 0;
    sDescription := 'Elemental density of Cu';
    sUnits := 'g/cm^3';
    sCaveat := '';
    bFound := TRUE;
ELSIF sName = 'Zn' THEN
    fValue := 7.133; (* Units: g/cm^3 *)
    fUncertainty := 0;
    sDescription := 'Elemental density of Zn';
    sUnits := 'g/cm^3';
    sCaveat := 'T=25';
    bFound := TRUE;
ELSIF sName = 'Ga' THEN
    fValue := 5.904; (* Units: g/cm^3 *)
    fUncertainty := 0;
    sDescription := 'Elemental density of Ga';
    sUnits := 'g/cm^3';
    sCaveat := 'T=29.6';
    bFound := TRUE;
ELSIF sName = 'Ge' THEN
    fValue := 5.323; (* Units: g/cm^3 *)
    fUncertainty := 0;
    sDescription := 'Elemental density of Ge';
    sUnits := 'g/cm^3';
    sCaveat := 'T=25';
    bFound := TRUE;
ELSIF sName = 'As' THEN
    fValue := 5.73; (* Units: g/cm^3 *)
    fUncertainty := 0;
    sDescription := 'Elemental density of As';
    sUnits := 'g/cm^3';
    sCaveat := '';
    bFound := TRUE;
ELSIF sName = 'Se' THEN
    fValue := 4.79; (* Units: g/cm^3 *)
    fUncertainty := 0;
    sDescription := 'Elemental density of Se';
    sUnits := 'g/cm^3';
    sCaveat := '';
    bFound := TRUE;
ELSIF sName = 'Br' THEN
    fValue := 3.12; (* Units: g/cm^3 *)
    fUncertainty := 0;
    sDescription := 'Elemental density of Br';
    sUnits := 'g/cm^3';
    sCaveat := '';
    bFound := TRUE;
ELSIF sName = 'Kr' THEN
    fValue := 2.16; (* Units: g/cm^3 *)
    fUncertainty := 0;
    sDescription := 'Elemental density of Kr';
    sUnits := 'g/cm^3';
    sCaveat := 'T=-153.22';
    bFound := TRUE;
ELSIF sName = 'Rb' THEN
    fValue := 1.532; (* Units: g/cm^3 *)
    fUncertainty := 0;
    sDescription := 'Elemental density of Rb';
    sUnits := 'g/cm^3';
    sCaveat := '';
    bFound := TRUE;
ELSIF sName = 'Sr' THEN
    fValue := 2.54; (* Units: g/cm^3 *)
    fUncertainty := 0;
    sDescription := 'Elemental density of Sr';
    sUnits := 'g/cm^3';
    sCaveat := '';
    bFound := TRUE;
ELSIF sName = 'Y' THEN
    fValue := 4.469; (* Units: g/cm^3 *)
    fUncertainty := 0;
    sDescription := 'Elemental density of Y';
    sUnits := 'g/cm^3';
    sCaveat := 'T=25';
    bFound := TRUE;
ELSIF sName = 'Zr' THEN
    fValue := 6.506; (* Units: g/cm^3 *)
    fUncertainty := 0;
    sDescription := 'Elemental density of Zr';
    sUnits := 'g/cm^3';
    sCaveat := '';
    bFound := TRUE;
ELSIF sName = 'Nb' THEN
    fValue := 8.57; (* Units: g/cm^3 *)
    fUncertainty := 0;
    sDescription := 'Elemental density of Nb';
    sUnits := 'g/cm^3';
    sCaveat := '';
    bFound := TRUE;
ELSIF sName = 'Mo' THEN
    fValue := 10.22; (* Units: g/cm^3 *)
    fUncertainty := 0;
    sDescription := 'Elemental density of Mo';
    sUnits := 'g/cm^3';
    sCaveat := '';
    bFound := TRUE;
ELSIF sName = 'Tc' THEN
    fValue := 11.5; (* Units: g/cm^3 *)
    fUncertainty := 0;
    sDescription := 'Elemental density of Tc';
    sUnits := 'g/cm^3';
    sCaveat := 'calculated';
    bFound := TRUE;
ELSIF sName = 'Ru' THEN
    fValue := 12.41; (* Units: g/cm^3 *)
    fUncertainty := 0;
    sDescription := 'Elemental density of Ru';
    sUnits := 'g/cm^3';
    sCaveat := '';
    bFound := TRUE;
ELSIF sName = 'Rh' THEN
    fValue := 12.41; (* Units: g/cm^3 *)
    fUncertainty := 0;
    sDescription := 'Elemental density of Rh';
    sUnits := 'g/cm^3';
    sCaveat := '';
    bFound := TRUE;
ELSIF sName = 'Pd' THEN
    fValue := 12.02; (* Units: g/cm^3 *)
    fUncertainty := 0;
    sDescription := 'Elemental density of Pd';
    sUnits := 'g/cm^3';
    sCaveat := '';
    bFound := TRUE;
ELSIF sName = 'Ag' THEN
    fValue := 10.5; (* Units: g/cm^3 *)
    fUncertainty := 0;
    sDescription := 'Elemental density of Ag';
    sUnits := 'g/cm^3';
    sCaveat := '';
    bFound := TRUE;
ELSIF sName = 'Cd' THEN
    fValue := 8.65; (* Units: g/cm^3 *)
    fUncertainty := 0;
    sDescription := 'Elemental density of Cd';
    sUnits := 'g/cm^3';
    sCaveat := '';
    bFound := TRUE;
ELSIF sName = 'In' THEN
    fValue := 7.31; (* Units: g/cm^3 *)
    fUncertainty := 0;
    sDescription := 'Elemental density of In';
    sUnits := 'g/cm^3';
    sCaveat := '';
    bFound := TRUE;
ELSIF sName = 'Sn' THEN
    fValue := 7.31; (* Units: g/cm^3 *)
    fUncertainty := 0;
    sDescription := 'Elemental density of Sn';
    sUnits := 'g/cm^3';
    sCaveat := '';
    bFound := TRUE;
ELSIF sName = 'Sb' THEN
    fValue := 6.691; (* Units: g/cm^3 *)
    fUncertainty := 0;
    sDescription := 'Elemental density of Sb';
    sUnits := 'g/cm^3';
    sCaveat := '';
    bFound := TRUE;
ELSIF sName = 'Te' THEN
    fValue := 6.24; (* Units: g/cm^3 *)
    fUncertainty := 0;
    sDescription := 'Elemental density of Te';
    sUnits := 'g/cm^3';
    sCaveat := '';
    bFound := TRUE;
ELSIF sName = 'I' THEN
    fValue := 4.93; (* Units: g/cm^3 *)
    fUncertainty := 0;
    sDescription := 'Elemental density of I';
    sUnits := 'g/cm^3';
    sCaveat := '';
    bFound := TRUE;
ELSIF sName = 'Xe' THEN
    fValue := 3.52; (* Units: g/cm^3 *)
    fUncertainty := 0;
    sDescription := 'Elemental density of Xe';
    sUnits := 'g/cm^3';
    sCaveat := 'T=-108.12';
    bFound := TRUE;
ELSIF sName = 'Cs' THEN
    fValue := 1.873; (* Units: g/cm^3 *)
    fUncertainty := 0;
    sDescription := 'Elemental density of Cs';
    sUnits := 'g/cm^3';
    sCaveat := '';
    bFound := TRUE;
ELSIF sName = 'Ba' THEN
    fValue := 3.5; (* Units: g/cm^3 *)
    fUncertainty := 0;
    sDescription := 'Elemental density of Ba';
    sUnits := 'g/cm^3';
    sCaveat := '';
    bFound := TRUE;
ELSIF sName = 'La' THEN
    fValue := 6.145; (* Units: g/cm^3 *)
    fUncertainty := 0;
    sDescription := 'Elemental density of La';
    sUnits := 'g/cm^3';
    sCaveat := 'T=25';
    bFound := TRUE;
ELSIF sName = 'Ce' THEN
    fValue := 6.77; (* Units: g/cm^3 *)
    fUncertainty := 0;
    sDescription := 'Elemental density of Ce';
    sUnits := 'g/cm^3';
    sCaveat := 'T=25';
    bFound := TRUE;
ELSIF sName = 'Pr' THEN
    fValue := 6.773; (* Units: g/cm^3 *)
    fUncertainty := 0;
    sDescription := 'Elemental density of Pr';
    sUnits := 'g/cm^3';
    sCaveat := '';
    bFound := TRUE;
ELSIF sName = 'Nd' THEN
    fValue := 7.008; (* Units: g/cm^3 *)
    fUncertainty := 0;
    sDescription := 'Elemental density of Nd';
    sUnits := 'g/cm^3';
    sCaveat := 'T=25';
    bFound := TRUE;
ELSIF sName = 'Pm' THEN
    fValue := 7.264; (* Units: g/cm^3 *)
    fUncertainty := 0;
    sDescription := 'Elemental density of Pm';
    sUnits := 'g/cm^3';
    sCaveat := 'T=25';
    bFound := TRUE;
ELSIF sName = 'Sm' THEN
    fValue := 7.52; (* Units: g/cm^3 *)
    fUncertainty := 0;
    sDescription := 'Elemental density of Sm';
    sUnits := 'g/cm^3';
    sCaveat := 'T=25';
    bFound := TRUE;
ELSIF sName = 'Eu' THEN
    fValue := 5.244; (* Units: g/cm^3 *)
    fUncertainty := 0;
    sDescription := 'Elemental density of Eu';
    sUnits := 'g/cm^3';
    sCaveat := 'T=25';
    bFound := TRUE;
ELSIF sName = 'Gd' THEN
    fValue := 7.901; (* Units: g/cm^3 *)
    fUncertainty := 0;
    sDescription := 'Elemental density of Gd';
    sUnits := 'g/cm^3';
    sCaveat := 'T=25';
    bFound := TRUE;
ELSIF sName = 'Tb' THEN
    fValue := 8.23; (* Units: g/cm^3 *)
    fUncertainty := 0;
    sDescription := 'Elemental density of Tb';
    sUnits := 'g/cm^3';
    sCaveat := '';
    bFound := TRUE;
ELSIF sName = 'Dy' THEN
    fValue := 8.551; (* Units: g/cm^3 *)
    fUncertainty := 0;
    sDescription := 'Elemental density of Dy';
    sUnits := 'g/cm^3';
    sCaveat := 'T=25';
    bFound := TRUE;
ELSIF sName = 'Ho' THEN
    fValue := 8.795; (* Units: g/cm^3 *)
    fUncertainty := 0;
    sDescription := 'Elemental density of Ho';
    sUnits := 'g/cm^3';
    sCaveat := 'T=25';
    bFound := TRUE;
ELSIF sName = 'Er' THEN
    fValue := 9.066; (* Units: g/cm^3 *)
    fUncertainty := 0;
    sDescription := 'Elemental density of Er';
    sUnits := 'g/cm^3';
    sCaveat := 'T=25';
    bFound := TRUE;
ELSIF sName = 'Tm' THEN
    fValue := 9.321; (* Units: g/cm^3 *)
    fUncertainty := 0;
    sDescription := 'Elemental density of Tm';
    sUnits := 'g/cm^3';
    sCaveat := 'T=25';
    bFound := TRUE;
ELSIF sName = 'Yb' THEN
    fValue := 6.966; (* Units: g/cm^3 *)
    fUncertainty := 0;
    sDescription := 'Elemental density of Yb';
    sUnits := 'g/cm^3';
    sCaveat := '';
    bFound := TRUE;
ELSIF sName = 'Lu' THEN
    fValue := 9.841; (* Units: g/cm^3 *)
    fUncertainty := 0;
    sDescription := 'Elemental density of Lu';
    sUnits := 'g/cm^3';
    sCaveat := 'T=25';
    bFound := TRUE;
ELSIF sName = 'Hf' THEN
    fValue := 13.31; (* Units: g/cm^3 *)
    fUncertainty := 0;
    sDescription := 'Elemental density of Hf';
    sUnits := 'g/cm^3';
    sCaveat := '';
    bFound := TRUE;
ELSIF sName = 'Ta' THEN
    fValue := 16.654; (* Units: g/cm^3 *)
    fUncertainty := 0;
    sDescription := 'Elemental density of Ta';
    sUnits := 'g/cm^3';
    sCaveat := '';
    bFound := TRUE;
ELSIF sName = 'W' THEN
    fValue := 19.3; (* Units: g/cm^3 *)
    fUncertainty := 0;
    sDescription := 'Elemental density of W';
    sUnits := 'g/cm^3';
    sCaveat := '';
    bFound := TRUE;
ELSIF sName = 'Re' THEN
    fValue := 21.02; (* Units: g/cm^3 *)
    fUncertainty := 0;
    sDescription := 'Elemental density of Re';
    sUnits := 'g/cm^3';
    sCaveat := '';
    bFound := TRUE;
ELSIF sName = 'Os' THEN
    fValue := 22.57; (* Units: g/cm^3 *)
    fUncertainty := 0;
    sDescription := 'Elemental density of Os';
    sUnits := 'g/cm^3';
    sCaveat := '';
    bFound := TRUE;
ELSIF sName = 'Ir' THEN
    fValue := 22.42; (* Units: g/cm^3 *)
    fUncertainty := 0;
    sDescription := 'Elemental density of Ir';
    sUnits := 'g/cm^3';
    sCaveat := 'T=17';
    bFound := TRUE;
ELSIF sName = 'Pt' THEN
    fValue := 21.45; (* Units: g/cm^3 *)
    fUncertainty := 0;
    sDescription := 'Elemental density of Pt';
    sUnits := 'g/cm^3';
    sCaveat := '';
    bFound := TRUE;
ELSIF sName = 'Au' THEN
    fValue := 19.3; (* Units: g/cm^3 *)
    fUncertainty := 0;
    sDescription := 'Elemental density of Au';
    sUnits := 'g/cm^3';
    sCaveat := 'approximate';
    bFound := TRUE;
ELSIF sName = 'Hg' THEN
    fValue := 13.546; (* Units: g/cm^3 *)
    fUncertainty := 0;
    sDescription := 'Elemental density of Hg';
    sUnits := 'g/cm^3';
    sCaveat := '';
    bFound := TRUE;
ELSIF sName = 'Tl' THEN
    fValue := 11.85; (* Units: g/cm^3 *)
    fUncertainty := 0;
    sDescription := 'Elemental density of Tl';
    sUnits := 'g/cm^3';
    sCaveat := '';
    bFound := TRUE;
ELSIF sName = 'Pb' THEN
    fValue := 11.35; (* Units: g/cm^3 *)
    fUncertainty := 0;
    sDescription := 'Elemental density of Pb';
    sUnits := 'g/cm^3';
    sCaveat := '';
    bFound := TRUE;
ELSIF sName = 'Bi' THEN
    fValue := 9.747; (* Units: g/cm^3 *)
    fUncertainty := 0;
    sDescription := 'Elemental density of Bi';
    sUnits := 'g/cm^3';
    sCaveat := '';
    bFound := TRUE;
ELSIF sName = 'Po' THEN
    fValue := 9.32; (* Units: g/cm^3 *)
    fUncertainty := 0;
    sDescription := 'Elemental density of Po';
    sUnits := 'g/cm^3';
    sCaveat := '';
    bFound := TRUE;
ELSIF sName = 'Th' THEN
    fValue := 11.72; (* Units: g/cm^3 *)
    fUncertainty := 0;
    sDescription := 'Elemental density of Th';
    sUnits := 'g/cm^3';
    sCaveat := '';
    bFound := TRUE;
ELSIF sName = 'Pa' THEN
    fValue := 15.37; (* Units: g/cm^3 *)
    fUncertainty := 0;
    sDescription := 'Elemental density of Pa';
    sUnits := 'g/cm^3';
    sCaveat := 'calculated';
    bFound := TRUE;
ELSIF sName = 'U' THEN
    fValue := 18.95; (* Units: g/cm^3 *)
    fUncertainty := 0;
    sDescription := 'Elemental density of U';
    sUnits := 'g/cm^3';
    sCaveat := 'approximate';
    bFound := TRUE;
ELSIF sName = 'Np' THEN
    fValue := 20.25; (* Units: g/cm^3 *)
    fUncertainty := 0;
    sDescription := 'Elemental density of Np';
    sUnits := 'g/cm^3';
    sCaveat := '';
    bFound := TRUE;
ELSIF sName = 'Pu' THEN
    fValue := 19.84; (* Units: g/cm^3 *)
    fUncertainty := 0;
    sDescription := 'Elemental density of Pu';
    sUnits := 'g/cm^3';
    sCaveat := 'T=25';
    bFound := TRUE;
ELSIF sName = 'Am' THEN
    fValue := 13.67; (* Units: g/cm^3 *)
    fUncertainty := 0;
    sDescription := 'Elemental density of Am';
    sUnits := 'g/cm^3';
    sCaveat := '';
    bFound := TRUE;
ELSIF sName = 'Cm' THEN
    fValue := 13.51; (* Units: g/cm^3 *)
    fUncertainty := 0;
    sDescription := 'Elemental density of Cm';
    sUnits := 'g/cm^3';
    sCaveat := 'calculated';
    bFound := TRUE;
ELSIF sName = 'Bk' THEN
    fValue := 14; (* Units: g/cm^3 *)
    fUncertainty := 0;
    sDescription := 'Elemental density of Bk';
    sUnits := 'g/cm^3';
    sCaveat := 'estimated';
    bFound := TRUE;
ELSE
    bFound := FALSE;
    fValue := 0;
    fUncertainty := 0;
    sDescription := '';
    sUnits := '';
    sCaveat := '';
END_IF

END_FUNCTION_BLOCK

// ---- Tests/FB_ScatteringFactorLookupCXRO_Test.TcPOU

FUNCTION_BLOCK FB_ScatteringFactorLookupCXRO_Test EXTENDS TcUnit.FB_TestSuite
VAR
END_VAR


GivenValidInputsExpectCorrectResult();


METHOD PRIVATE GivenValidInputsExpectCorrectResult
VAR_INST
    fResult : LREAL;
    bError : BOOL;
    sErrorMsg : T_MaxString;
    fbScatteringFactorLookupCXRO : FB_ScatteringFactorLookupCXRO;
END_VAR

TEST('GivenValidInputsExpectCorrectResult');

fbScatteringFactorLookupCXRO.GetScatteringFactor(
    sMaterialName := 'C',
    fPhotonEnergy_eV := 10000,
    f2 => fResult,
    bError => bError,
    sErrorMsg => sErrorMsg
);

AssertEquals_BOOL(
    Expected := FALSE,
    Actual := bError,
    Message := 'Expected no error'
);

AssertEquals_STRING(
    Expected := '',
    Actual := sErrorMsg,
    Message := 'Expected empty error string'
);

AssertEquals_LREAL(
    Expected := 0.0058932368755846573,
    Actual := fResult,
    Delta := 1e-9,
    Message := 'Incorrect result.'
);

TEST_FINISHED();
END_METHOD

END_FUNCTION_BLOCK

// ---- POUs/FB_ScatteringFactorLookupCXRO.TcPOU

FUNCTION_BLOCK FB_ScatteringFactorLookupCXRO IMPLEMENTS I_ScatteringFactorLookup
VAR
    fbScatteringFactorLUT : FB_ScatteringFactorLUT;
END_VAR


METHOD FB_Init: BOOL
VAR_INPUT
    bInitRetains: BOOL; // TRUE: the retain variables are initialized (reset warm / reset cold)
    bInCopyCode: BOOL;  // TRUE: the instance will be copied to the copy code afterward (online change)
END_VAR

fbScatteringFactorLUT(
    sTableName := 'Ge',
    fEnergyEV := 10.0
);
END_METHOD


METHOD GetScatteringFactor
VAR_INPUT
    (* Chemical formula for the material as a string. *)
    sMaterialName	: T_MaxString;
    (* Photon energy in eV. *)
    fPhotonEnergy_eV	: LREAL;
END_VAR
VAR_OUTPUT
    f1 : LREAL;
    f2 : LREAL;
    bError : BOOL;
    sErrorMsg : T_MaxString;
END_VAR

THIS^.fbScatteringFactorLUT(
    sTableName := sMaterialName,
    fEnergyEV := fPhotonEnergy_eV,
    f1 => f1,
    f2 => f2,
    bError => bError
);

IF NOT THIS^.fbScatteringFactorLUT.bFound THEN
    sErrorMsg := 'Input photon energy not found in the lookup table.';
END_IF
END_METHOD


PROPERTY MaximumValidLookupPhotonEnergy_eV : LREAL
GET

MaximumValidLookupPhotonEnergy_eV := THIS^.fbScatteringFactorLUT.fTableLookupHigh;
END_GET
END_PROPERTY


PROPERTY MinimumValidLookupPhotonEnergy_eV : LREAL
GET

MinimumValidLookupPhotonEnergy_eV := THIS^.fbScatteringFactorLUT.fTableLookupLow;
END_GET
END_PROPERTY

END_FUNCTION_BLOCK

// ---- POUs/FB_ScatteringFactorLUT.TcPOU

(* WARNING: This file is auto-generated. Do not modify it.*)
FUNCTION_BLOCK FB_ScatteringFactorLUT
VAR_INPUT
    sTableName : STRING;
    fEnergyEV : LREAL;
END_VAR
VAR_OUTPUT
    f1 : LREAL;
    f2 : LREAL;
    bError : BOOL; (* Was the table name or data invalid? *)
    bFound : BOOL; (* Was the input found in the table? *)
    bDone : BOOL;  (* Has the FB finished? *)

    fTableLookupLow: LREAL; (* The lowest accepted lookup value. *)
    fTableLookupHigh: LREAL; (* The highest accepted lookup value. *)
END_VAR
VAR

    bInit : BOOL;
    iRowSize : UDINT;
    fRow1 : POINTER TO ARRAY[0..2] OF LREAL;
    fRow2 : POINTER TO ARRAY[0..2] OF LREAL;
    fEnergyEV_RowDelta : LREAL;

    iRowCount : UDINT;
    iRowIdx : UDINT;
    fSlope : LREAL;

    (* The data tables. These are Initialized on the first function block call. *)

    fTable_Ge : ARRAY[0..505, 0..2] OF LREAL;

    fTable_C : ARRAY[0..501, 0..2] OF LREAL;

    fTable_Al : ARRAY[0..503, 0..2] OF LREAL;

    fTable_Be : ARRAY[0..723, 0..2] OF LREAL;

    fTable_Si : ARRAY[0..755, 0..2] OF LREAL;

END_VAR


(* WARNING: This file is auto-generated. Do not modify it.*)

bError := FALSE;
bFound := FALSE;
bDone := FALSE;

IF NOT bInit THEN

